KUKA KRL program: MyProgram_228().src

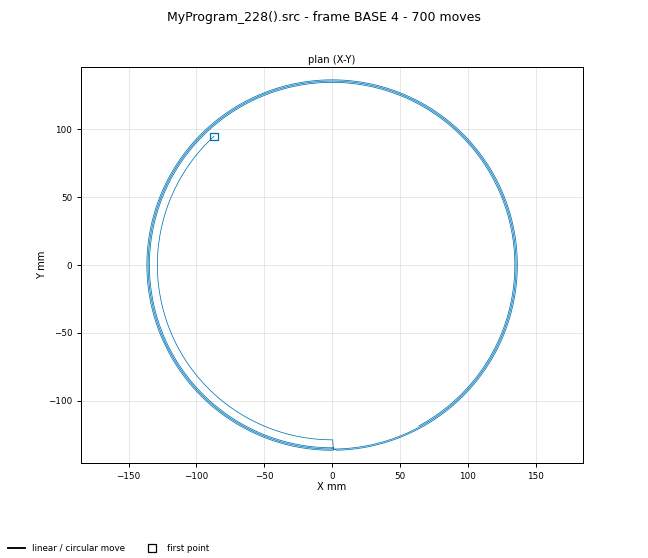
[picture p0: tool path of MyProgram_228().src in frame BASE 4, 700 of 700 moves have a stored position in this frame; points joined in program order, loops and branches not executed]
&ACCESS RVP
&REL 1
&PARAM TEMPLATE = C:\KRC\Roboter\Template\vorgabe
&PARAM EDITMASK = *
DEF MyProgram_228()
; ---- Setting reference (Base) ----
$BASE = BASE_DATA[4]

; --------------------------
; ---- Setting tool (TCP) ----
$TOOL = TOOL_DATA[3]
; --------------------------

$VEL.CP = VEL_APROX_PRINT
Startdeposition()
$VEL.CP = VEL_PRINT
LIN {X -87.249,Y 94.7644,Z 156,A 131.7376,B 16.1467,C -0.3808,E1 16.0419,E2 317.28} C_DIS
LIN {X -90.1231,Y 92.0354,Z 156,A 133.506,B 16.1468,C -0.3771,E1 16.0384,E2 315.5131} C_DIS
LIN {X -93.2907,Y 88.8233,Z 156,A 135.5438,B 16.1468,C -0.3735,E1 16.0344,E2 313.4743} C_DIS
LIN {X -95.9677,Y 85.9237,Z 156,A 137.2975,B 16.147,C -0.3694,E1 16.0311,E2 311.7231} C_DIS
LIN {X -98.5652,Y 82.9313,Z 156,A 139.0194,B 16.1471,C -0.364,E1 16.028,E2 310.008} C_DIS
LIN {X -101.0601,Y 79.8729,Z 156,A 140.9035,B 16.1471,C -0.3635,E1 16.0247,E2 308.1116} C_DIS
LIN {X -103.7403,Y 76.3586,Z 156,A 142.847,B 16.1472,C -0.3579,E1 16.0215,E2 306.1732} C_DIS
LIN {X -106.2189,Y 72.8714,Z 156,A 144.716,B 16.1474,C -0.352,E1 16.0185,E2 304.3107} C_DIS
LIN {X -108.2169,Y 69.8706,Z 156,A 146.2635,B 16.1474,C -0.3462,E1 16.0161,E2 302.7718} C_DIS
LIN {X -109.8979,Y 67.195,Z 156,A 147.6521,B 16.1476,C -0.342,E1 16.0141,E2 301.3869} C_DIS
LIN {X -111.2983,Y 64.8499,Z 156,A 148.8967,B 16.1476,C -0.3396,E1 16.0123,E2 300.1406} C_DIS
LIN {X -112.8404,Y 62.1274,Z 156,A 150.3075,B 16.1476,C -0.3364,E1 16.0104,E2 298.7295} C_DIS
LIN {X -114.5112,Y 58.9894,Z 156,A 151.8787,B 16.1478,C -0.3318,E1 16.0084,E2 297.1616} C_DIS
LIN {X -115.8793,Y 56.2567,Z 156,A 153.2802,B 16.1478,C -0.3292,E1 16.0066,E2 295.7572} C_DIS
LIN {X -117.1898,Y 53.4711,Z 156,A 154.6946,B 16.1478,C -0.3267,E1 16.005,E2 294.3395} C_DIS
LIN {X -118.5677,Y 50.3434,Z 156,A 156.1834,B 16.148,C -0.3214,E1 16.0033,E2 292.8564} C_DIS
LIN {X -119.7652,Y 47.4248,Z 156,A 157.6082,B 16.148,C -0.3181,E1 16.0019,E2 291.4311} C_DIS
LIN {X -120.8905,Y 44.4777,Z 156,A 159.166,B 16.148,C -0.3185,E1 16.0003,E2 289.8575} C_DIS
LIN {X -122.1722,Y 40.8189,Z 156,A 160.8434,B 16.1482,C -0.3121,E1 15.9988,E2 288.1877} C_DIS
LIN {X -123.2669,Y 37.3845,Z 156,A 162.4226,B 16.1482,C -0.3067,E1 15.9975,E2 286.6135} C_DIS
LIN {X -124.267,Y 33.9193,Z 156,A 164.0055,B 16.1484,C -0.3013,E1 15.9963,E2 285.0354} C_DIS
LIN {X -125.2204,Y 30.2007,Z 156,A 165.4905,B 16.1486,C -0.2898,E1 15.9953,E2 283.5781} C_DIS
LIN {X -125.7812,Y 27.7795,Z 156,A 166.7692,B 16.1486,C -0.2915,E1 15.9945,E2 282.2811} C_DIS
LIN {X -126.4236,Y 24.6901,Z 156,A 168.1468,B 16.1486,C -0.2865,E1 15.9938,E2 280.9084} C_DIS
LIN {X -126.9922,Y 21.5728,Z 156,A 169.6871,B 16.1486,C -0.2861,E1 15.993,E2 279.355} C_DIS
LIN {X -127.4822,Y 18.4562,Z 156,A 170.9529,B 16.1488,C -0.2779,E1 15.9925,E2 278.1069} C_DIS
LIN {X -127.8958,Y 15.3281,Z 156,A 172.6093,B 16.1488,C -0.2809,E1 15.9919,E2 276.4233} C_DIS
LIN {X -128.3353,Y 11.0629,Z 156,A 174.5297,B 16.1488,C -0.2755,E1 15.9914,E2 274.504} C_DIS
LIN {X -128.5967,Y 7.4451,Z 156,A 176.2254,B 16.1488,C -0.273,E1 15.9911,E2 272.801} C_DIS
LIN {X -128.7414,Y 4.2996,Z 156,A 177.5163,B 16.149,C -0.2655,E1 15.991,E2 271.5246} C_DIS
LIN {X -128.8029,Y 1.5734,Z 156,A 178.8128,B 16.149,C -0.2643,E1 15.9909,E2 270.22} C_DIS
LIN {X -128.8028,Y -1.5789,Z 156,A -179.8543,B 16.149,C -0.258,E1 15.9909,E2 268.8969} C_DIS
LIN {X -128.7239,Y -4.7473,Z 156,A -178.4414,B 16.1492,C -0.2538,E1 15.991,E2 267.4854} C_DIS
LIN {X -128.5687,Y -7.8985,Z 156,A -176.9705,B 16.1492,C -0.2515,E1 15.9913,E2 266.0085} C_DIS
LIN {X -128.2352,Y -12.1673,Z 156,A -175.3618,B 16.1494,C -0.2372,E1 15.9916,E2 264.4362} C_DIS
LIN {X -127.899,Y -15.3015,Z 156,A -173.6271,B 16.1494,C -0.2426,E1 15.9922,E2 262.665} C_DIS
LIN {X -127.4183,Y -18.9032,Z 156,A -172.0698,B 16.1494,C -0.2361,E1 15.9928,E2 261.1165} C_DIS
LIN {X -126.8381,Y -22.4593,Z 156,A -170.5916,B 16.1495,C -0.2277,E1 15.9935,E2 259.6545} C_DIS
LIN {X -126.2498,Y -25.5591,Z 156,A -169.1609,B 16.1495,C -0.2243,E1 15.9942,E2 258.2223} C_DIS
LIN {X -125.5776,Y -28.6793,Z 156,A -167.594,B 16.1495,C -0.2245,E1 15.9952,E2 256.6402} C_DIS
LIN {X -124.6725,Y -32.3966,Z 156,A -165.7419,B 16.1495,C -0.2239,E1 15.9965,E2 254.7727} C_DIS
LIN {X -123.7153,Y -35.873,Z 156,A -164.1536,B 16.1497,C -0.2188,E1 15.9977,E2 253.1879} C_DIS
LIN {X -122.6587,Y -39.3328,Z 156,A -162.6301,B 16.1497,C -0.2117,E1 15.9989,E2 251.676} C_DIS
LIN {X -121.65,Y -42.3498,Z 156,A -161.112,B 16.1497,C -0.2107,E1 16.0003,E2 250.1475} C_DIS
LIN {X -120.177,Y -46.3659,Z 156,A -159.2834,B 16.1499,C -0.2032,E1 16.0021,E2 248.3295} C_DIS
LIN {X -119.0055,Y -49.2954,Z 156,A -157.8691,B 16.1499,C -0.1997,E1 16.0036,E2 246.9153} C_DIS
LIN {X -117.7369,Y -52.2526,Z 156,A -156.4462,B 16.1499,C -0.1955,E1 16.0052,E2 245.4948} C_DIS
LIN {X -116.4498,Y -55.0627,Z 156,A -155.0417,B 16.1499,C -0.1927,E1 16.0068,E2 244.0882} C_DIS
LIN {X -114.9305,Y -58.1657,Z 156,A -153.4439,B 16.15,C -0.1904,E1 16.0088,E2 242.4848} C_DIS
LIN {X -113.3903,Y -61.1175,Z 156,A -151.9893,B 16.15,C -0.1857,E1 16.0107,E2 241.0347} C_DIS
LIN {X -111.7243,Y -64.113,Z 156,A -150.489,B 16.1501,C -0.1811,E1 16.0128,E2 239.5386} C_DIS
LIN {X -110.1684,Y -66.7504,Z 156,A -148.9834,B 16.1501,C -0.1819,E1 16.015,E2 238.0175} C_DIS
LIN {X -107.9795,Y -70.2361,Z 156,A -147.2344,B 16.1501,C -0.1749,E1 16.0176,E2 236.2795} C_DIS
LIN {X -105.9806,Y -73.2185,Z 156,A -145.4796,B 16.1501,C -0.1758,E1 16.0204,E2 234.5076} C_DIS
LIN {X -103.4626,Y -76.7348,Z 156,A -143.5723,B 16.1502,C -0.1707,E1 16.0235,E2 232.6037} C_DIS
LIN {X -100.9438,Y -80.0194,Z 156,A -141.6939,B 16.1502,C -0.1676,E1 16.0267,E2 230.7223} C_DIS
LIN {X -98.0535,Y -83.5357,Z 156,A -139.6814,B 16.1503,C -0.1627,E1 16.0303,E2 228.7126} C_DIS
LIN {X -95.448,Y -86.5006,Z 156,A -137.9263,B 16.1503,C -0.1589,E1 16.0336,E2 226.9587} C_DIS
LIN {X -93.1464,Y -88.9743,Z 156,A -136.4044,B 16.1503,C -0.1563,E1 16.0365,E2 225.4355} C_DIS
LIN {X -89.9537,Y -92.2016,Z 156,A -134.316,B 16.1503,C -0.1543,E1 16.0407,E2 223.3401} C_DIS
LIN {X -86.9226,Y -95.0644,Z 156,A -132.4884,B 16.1504,C -0.1498,E1 16.0444,E2 221.5167} C_DIS
LIN {X -83.9704,Y -97.6815,Z 156,A -130.7347,B 16.1504,C -0.1465,E1 16.0481,E2 219.7639} C_DIS
LIN {X -80.6634,Y -100.4299,Z 156,A -128.8883,B 16.1505,C -0.141,E1 16.0521,E2 217.9261} C_DIS
LIN {X -77.64,Y -102.7848,Z 156,A -127.2105,B 16.1505,C -0.1373,E1 16.0558,E2 216.2521} C_DIS
LIN {X -74.5444,Y -105.0521,Z 156,A -125.3895,B 16.1505,C -0.138,E1 16.0599,E2 214.4185} C_DIS
LIN {X -71.1886,Y -107.3547,Z 156,A -123.5938,B 16.1505,C -0.1347,E1 16.0641,E2 212.625} C_DIS
LIN {X -68.5545,Y -109.0551,Z 156,A -122.2704,B 16.1505,C -0.1304,E1 16.0672,E2 211.3103} C_DIS
LIN {X -66.2577,Y -110.466,Z 156,A -121.0601,B 16.1505,C -0.129,E1 16.0701,E2 210.099} C_DIS
LIN {X -63.4903,Y -112.0795,Z 156,A -119.6307,B 16.1506,C -0.1272,E1 16.0735,E2 208.6694} C_DIS
LIN {X -60.7258,Y -113.6008,Z 156,A -118.1094,B 16.1506,C -0.129,E1 16.0773,E2 207.1345} C_DIS
LIN {X -57.5236,Y -115.2544,Z 156,A -116.6236,B 16.1506,C -0.1234,E1 16.081,E2 205.6627} C_DIS
LIN {X -54.6526,Y -116.6434,Z 156,A -115.249,B 16.1506,C -0.1203,E1 16.0844,E2 204.2934} C_DIS
LIN {X -51.8174,Y -117.931,Z 156,A -113.8147,B 16.1506,C -0.1203,E1 16.0881,E2 202.8535} C_DIS
LIN {X -48.9638,Y -119.1439,Z 156,A -112.4154,B 16.1506,C -0.1196,E1 16.0917,E2 201.4519} C_DIS
LIN {X -46.1238,Y -120.2711,Z 156,A -111.0448,B 16.1506,C -0.1187,E1 16.0953,E2 200.0799} C_DIS
LIN {X -42.3323,Y -121.6561,Z 156,A -109.172,B 16.1506,C -0.1196,E1 16.1002,E2 198.198} C_DIS
LIN {X -38.3136,Y -122.9825,Z 156,A -107.2264,B 16.1506,C -0.1201,E1 16.1054,E2 196.2449} C_DIS
LIN {X -35.3586,Y -123.8647,Z 156,A -105.9028,B 16.1506,C -0.1176,E1 16.109,E2 194.9268} C_DIS
LIN {X -32.4047,Y -124.6704,Z 156,A -104.4449,B 16.1506,C -0.1198,E1 16.1129,E2 193.4574} C_DIS
LIN {X -29.3446,Y -125.4257,Z 156,A -103.2191,B 16.1507,C -0.1134,E1 16.1162,E2 192.2521} C_DIS
LIN {X -26.6975,Y -126.0148,Z 156,A -101.9339,B 16.1507,C -0.1154,E1 16.1197,E2 190.9574} C_DIS
LIN {X -23.3363,Y -126.6811,Z 156,A -100.4229,B 16.1507,C -0.1143,E1 16.1239,E2 189.4476} C_DIS
LIN {X -20.059,Y -127.2401,Z 156,A -98.9484,B 16.1507,C -0.1137,E1 16.1279,E2 187.9731} C_DIS
LIN {X -15.4689,Y -127.879,Z 156,A -97.1029,B 16.1507,C -0.1062,E1 16.133,E2 186.1525} C_DIS
LIN {X -12.6065,Y -128.1931,Z 156,A -95.5324,B 16.1507,C -0.1154,E1 16.1374,E2 184.5474} C_DIS
LIN {X -9.0242,Y -128.4951,Z 156,A -94.0776,B 16.1507,C -0.1106,E1 16.1414,E2 183.109} C_DIS
LIN {X -5.1896,Y -128.7067,Z 156,A -92.6012,B 16.1507,C -0.1031,E1 16.1455,E2 181.6591} C_DIS
LIN {X -2.7134,Y -128.7839,Z 156,A -91.3422,B 16.1507,C -0.1083,E1 16.1491,E2 180.3813} C_DIS
LIN {X 0.4448,Y -128.8107,Z 156,A -89.7625,B 16.1507,C -0.1142,E1 16.1535,E2 178.7802} C_DIS
LIN {X 0.4448,Y -128.8107,Z 156,A -89.7625,B 16.1507,C -0.1142,E1 16.1535,E2 178.7802} C_DIS
Enddeposition()
LIN {X 0.9577,Y -136.4876,Z 157,A -93.1618,B 24.9717,C -1.2298,E1 24.9996,E2 179.8882} C_DIS
Startdeposition()
$VEL.CP = VEL_PRINT
LIN {X -4.793,Y -136.4624,Z 157,A -95.2992,B 24.9711,C -1.2432,E1 24.9937,E2 181.994} C_DIS
LIN {X -11.5417,Y -136.0568,Z 157,A -97.812,B 24.9702,C -1.2606,E1 24.9869,E2 184.4665} C_DIS
LIN {X -17.4629,Y -135.4244,Z 157,A -100.4347,B 24.9705,C -1.2541,E1 24.9795,E2 187.106} C_DIS
LIN {X -22.0632,Y -134.7517,Z 157,A -102.641,B 24.9712,C -1.241,E1 24.9733,E2 189.3454} C_DIS
LIN {X -25.4466,Y -134.1534,Z 157,A -104.0634,B 24.9711,C -1.2426,E1 24.9694,E2 190.7655} C_DIS
LIN {X -28.8158,Y -133.4701,Z 157,A -105.4664,B 24.971,C -1.2453,E1 24.9656,E2 192.1637} C_DIS
LIN {X -32.1255,Y -132.7124,Z 157,A -106.9209,B 24.971,C -1.2445,E1 24.9617,E2 193.6221} C_DIS
LIN {X -35.9393,Y -131.7329,Z 157,A -108.5566,B 24.971,C -1.2463,E1 24.9572,E2 195.2558} C_DIS
LIN {X -38.9621,Y -130.8698,Z 157,A -109.8853,B 24.9709,C -1.2468,E1 24.9537,E2 196.5856} C_DIS
LIN {X -42.1527,Y -129.8773,Z 157,A -111.2482,B 24.9707,C -1.25,E1 24.9501,E2 197.9434} C_DIS
LIN {X -44.9713,Y -128.9272,Z 157,A -112.5846,B 24.9709,C -1.2464,E1 24.9465,E2 199.2909} C_DIS
LIN {X -48.5684,Y -127.6173,Z 157,A -114.1394,B 24.9707,C -1.2506,E1 24.9425,E2 200.8389} C_DIS
LIN {X -51.6804,Y -126.3889,Z 157,A -115.5554,B 24.9707,C -1.2514,E1 24.9388,E2 202.2561} C_DIS
LIN {X -54.8493,Y -125.0464,Z 157,A -117.0748,B 24.9707,C -1.249,E1 24.9349,E2 203.7847} C_DIS
LIN {X -59.0833,Y -123.1006,Z 157,A -118.9953,B 24.9706,C -1.2532,E1 24.93,E2 205.7001} C_DIS
LIN {X -62.4726,Y -121.4169,Z 157,A -120.5555,B 24.9704,C -1.2567,E1 24.9261,E2 207.2562} C_DIS
LIN {X -65.2945,Y -119.9238,Z 157,A -122.0012,B 24.9706,C -1.253,E1 24.9225,E2 208.7148} C_DIS
LIN {X -69.2384,Y -117.6908,Z 157,A -123.9078,B 24.9705,C -1.2555,E1 24.9179,E2 210.621} C_DIS
LIN {X -73.2088,Y -115.2636,Z 157,A -125.7821,B 24.9701,C -1.2626,E1 24.9135,E2 212.4844} C_DIS
LIN {X -76.368,Y -113.1947,Z 157,A -127.4717,B 24.9703,C -1.2598,E1 24.9096,E2 214.1862} C_DIS
LIN {X -80.1611,Y -110.5408,Z 157,A -129.3474,B 24.97,C -1.2666,E1 24.9053,E2 216.0522} C_DIS
LIN {X -83.5476,Y -108.004,Z 157,A -131.1702,B 24.97,C -1.2674,E1 24.9012,E2 217.8796} C_DIS
LIN {X -87.0681,Y -105.1866,Z 157,A -133.1165,B 24.9699,C -1.2682,E1 24.897,E2 219.8314} C_DIS
LIN {X -90.2129,Y -102.5027,Z 157,A -134.8342,B 24.9697,C -1.2726,E1 24.8934,E2 221.5454} C_DIS
LIN {X -93.618,Y -99.402,Z 157,A -136.7917,B 24.9695,C -1.2753,E1 24.8894,E2 223.5043} C_DIS
LIN {X -96.6303,Y -96.4767,Z 157,A -138.5786,B 24.9695,C -1.2779,E1 24.8858,E2 225.2927} C_DIS
LIN {X -99.9068,Y -93.079,Z 157,A -140.4529,B 24.9689,C -1.2878,E1 24.8823,E2 227.1517} C_DIS
LIN {X -102.6938,Y -89.9952,Z 157,A -142.3091,B 24.969,C -1.2861,E1 24.8788,E2 229.0201} C_DIS
LIN {X -105.7402,Y -86.3949,Z 157,A -144.2944,B 24.9688,C -1.2906,E1 24.8752,E2 231.0039} C_DIS
LIN {X -108.6802,Y -82.6668,Z 157,A -146.2709,B 24.9685,C -1.2963,E1 24.8719,E2 232.9762} C_DIS
LIN {X -111.3396,Y -79.0489,Z 157,A -148.2093,B 24.9685,C -1.2984,E1 24.8687,E2 234.9191} C_DIS
LIN {X -113.7117,Y -75.5962,Z 157,A -149.8638,B 24.9679,C -1.3082,E1 24.8661,E2 236.5584} C_DIS
LIN {X -116.0225,Y -71.9991,Z 157,A -151.7512,B 24.9679,C -1.3082,E1 24.8633,E2 238.4552} C_DIS
LIN {X -118.1139,Y -68.5141,Z 157,A -153.3784,B 24.9675,C -1.3169,E1 24.861,E2 240.0702} C_DIS
LIN {X -120.101,Y -64.9689,Z 157,A -155.2095,B 24.9675,C -1.3153,E1 24.8585,E2 241.9147} C_DIS
LIN {X -124.9697,Y -55.025,Z 157,A -159.7494,B 24.9667,C -1.334,E1 24.8531,E2 246.4348} C_DIS
LIN {X -126.215,Y -52.1021,Z 157,A -161.0965,B 24.9665,C -1.3373,E1 24.8516,E2 247.7815} C_DIS
LIN {X -127.4612,Y -48.9743,Z 157,A -162.5034,B 24.9663,C -1.3418,E1 24.8502,E2 249.1855} C_DIS
LIN {X -128.6336,Y -45.8067,Z 157,A -164.0021,B 24.9663,C -1.3421,E1 24.8487,E2 250.6921} C_DIS
LIN {X -129.9079,Y -42.0571,Z 157,A -165.6808,B 24.966,C -1.3463,E1 24.8473,E2 252.3703} C_DIS
LIN {X -131.1342,Y -38.0593,Z 157,A -167.407,B 24.9657,C -1.3532,E1 24.8459,E2 254.09} C_DIS
LIN {X -132.2625,Y -33.9314,Z 157,A -169.2124,B 24.9654,C -1.3584,E1 24.8446,E2 255.8936} C_DIS
LIN {X -133.166,Y -30.1904,Z 157,A -170.8008,B 24.9651,C -1.3648,E1 24.8436,E2 257.476} C_DIS
LIN {X -133.9535,Y -26.4884,Z 157,A -172.5568,B 24.9653,C -1.3615,E1 24.8426,E2 259.2501} C_DIS
LIN {X -134.6769,Y -22.5112,Z 157,A -174.0908,B 24.9646,C -1.3751,E1 24.8419,E2 260.7609} C_DIS
LIN {X -135.1582,Y -19.4141,Z 157,A -175.4508,B 24.9645,C -1.3771,E1 24.8413,E2 262.1242} C_DIS
LIN {X -135.5862,Y -16.1562,Z 157,A -176.8171,B 24.9642,C -1.3823,E1 24.8408,E2 263.4865} C_DIS
LIN {X -135.9492,Y -12.7499,Z 157,A -178.3678,B 24.9642,C -1.3813,E1 24.8404,E2 265.0486} C_DIS
LIN {X -136.27,Y -8.6741,Z 157,A 179.954,B 24.9639,C -1.3888,E1 24.84,E2 266.719} C_DIS
LIN {X -136.4579,Y -4.9082,Z 157,A 178.3315,B 24.9637,C -1.392,E1 24.8399,E2 268.3437} C_DIS
LIN {X -136.5447,Y -0.6887,Z 157,A 176.589,B 24.9633,C -1.3993,E1 24.8398,E2 270.0794} C_DIS
LIN {X -136.503,Y 3.4288,Z 157,A 174.8401,B 24.9631,C -1.404,E1 24.8398,E2 271.8276} C_DIS
LIN {X -136.3626,Y 7.0678,Z 157,A 173.2663,B 24.9629,C -1.4068,E1 24.8401,E2 273.4042} C_DIS
LIN {X -136.0949,Y 11.0902,Z 157,A 171.5971,B 24.9626,C -1.4135,E1 24.8404,E2 275.0675} C_DIS
LIN {X -135.7642,Y 14.5853,Z 157,A 170.0652,B 24.9625,C -1.4155,E1 24.8408,E2 276.6038} C_DIS
LIN {X -135.2032,Y 19.0993,Z 157,A 168.2113,B 24.962,C -1.4245,E1 24.8415,E2 278.4473} C_DIS
LIN {X -134.686,Y 22.4568,Z 157,A 166.7957,B 24.9617,C -1.4297,E1 24.8421,E2 279.8589} C_DIS
LIN {X -134.0288,Y 26.0984,Z 157,A 165.0936,B 24.9618,C -1.4275,E1 24.843,E2 281.5765} C_DIS
LIN {X -133.0967,Y 30.4938,Z 157,A 163.3198,B 24.9612,C -1.4392,E1 24.8441,E2 283.3329} C_DIS
LIN {X -132.2919,Y 33.8157,Z 157,A 161.8501,B 24.961,C -1.4421,E1 24.8451,E2 284.8042} C_DIS
LIN {X -131.3195,Y 37.4195,Z 157,A 160.1661,B 24.961,C -1.4413,E1 24.8463,E2 286.4998} C_DIS
LIN {X -130.0192,Y 41.7086,Z 157,A 158.4113,B 24.9604,C -1.4536,E1 24.8478,E2 288.2353} C_DIS
LIN {X -128.769,Y 45.4274,Z 157,A 156.7633,B 24.9601,C -1.4588,E1 24.8493,E2 289.8805} C_DIS
LIN {X -127.6672,Y 48.4352,Z 157,A 155.4364,B 24.9599,C -1.4639,E1 24.8506,E2 291.2025} C_DIS
LIN {X -126.5043,Y 51.394,Z 157,A 154.0589,B 24.9597,C -1.466,E1 24.852,E2 292.5829} C_DIS
LIN {X -125.2431,Y 54.3945,Z 157,A 152.684,B 24.9595,C -1.4698,E1 24.8535,E2 293.9563} C_DIS
LIN {X -123.8056,Y 57.5917,Z 157,A 151.1641,B 24.9595,C -1.4719,E1 24.8553,E2 295.4794} C_DIS
LIN {X -122.2195,Y 60.8868,Z 157,A 149.6565,B 24.9591,C -1.4779,E1 24.8571,E2 296.9809} C_DIS
LIN {X -120.7158,Y 63.8151,Z 157,A 148.2867,B 24.9588,C -1.4827,E1 24.8589,E2 298.3466} C_DIS
LIN {X -118.6745,Y 67.5385,Z 157,A 146.4342,B 24.9588,C -1.4845,E1 24.8614,E2 300.2045} C_DIS
LIN {X -116.4781,Y 71.2598,Z 157,A 144.6247,B 24.9584,C -1.49,E1 24.864,E2 302.0102} C_DIS
LIN {X -114.272,Y 74.7472,Z 157,A 142.8205,B 24.9584,C -1.4914,E1 24.8667,E2 303.8202} C_DIS
LIN {X -111.805,Y 78.3892,Z 157,A 140.9498,B 24.9581,C -1.4954,E1 24.8697,E2 305.6906} C_DIS
LIN {X -108.9004,Y 82.3759,Z 157,A 138.7981,B 24.9581,C -1.4971,E1 24.8733,E2 307.8488} C_DIS
LIN {X -106.407,Y 85.5725,Z 157,A 137.1396,B 24.9576,C -1.5038,E1 24.8761,E2 309.4989} C_DIS
LIN {X -103.4241,Y 89.1545,Z 157,A 135.1904,B 24.9573,C -1.5094,E1 24.8796,E2 311.4439} C_DIS
LIN {X -100.3303,Y 92.6228,Z 157,A 133.2038,B 24.9571,C -1.5126,E1 24.8834,E2 313.4316} C_DIS
LIN {X -97.0811,Y 96.023,Z 157,A 131.3563,B 24.9565,C -1.5239,E1 24.8869,E2 315.2602} C_DIS
LIN {X -94.1868,Y 98.8633,Z 157,A 129.5508,B 24.9565,C -1.5228,E1 24.8906,E2 317.0758} C_DIS
LIN {X -90.8799,Y 101.9117,Z 157,A 127.6624,B 24.9563,C -1.5272,E1 24.8945,E2 318.9613} C_DIS
LIN {X -87.5334,Y 104.8001,Z 157,A 125.7574,B 24.9563,C -1.529,E1 24.8985,E2 320.8695} C_DIS
LIN {X -83.9195,Y 107.7158,Z 157,A 123.7927,B 24.956,C -1.5325,E1 24.9028,E2 322.8332} C_DIS
LIN {X -80.6451,Y 110.1884,Z 157,A 122.0698,B 24.9558,C -1.5361,E1 24.9067,E2 324.5536} C_DIS
LIN {X -76.8585,Y 112.8627,Z 157,A 120.1088,B 24.9556,C -1.5393,E1 24.9112,E2 326.5137} C_DIS
LIN {X -73.1617,Y 115.2933,Z 157,A 118.2561,B 24.9554,C -1.5431,E1 24.9155,E2 328.3633} C_DIS
LIN {X -68.7626,Y 117.9701,Z 157,A 116.1991,B 24.9548,C -1.5524,E1 24.9204,E2 330.4045} C_DIS
LIN {X -65.2408,Y 119.9531,Z 157,A 114.3542,B 24.9551,C -1.5479,E1 24.925,E2 332.2654} C_DIS
LIN {X -61.8376,Y 121.7401,Z 157,A 112.8706,B 24.9546,C -1.5572,E1 24.9286,E2 333.7308} C_DIS
LIN {X -58.5691,Y 123.3463,Z 157,A 111.3055,B 24.9546,C -1.5578,E1 24.9325,E2 335.2986} C_DIS
LIN {X -54.9799,Y 124.9899,Z 157,A 109.6879,B 24.9543,C -1.5623,E1 24.9366,E2 336.9095} C_DIS
LIN {X -51.8857,Y 126.3054,Z 157,A 108.2749,B 24.9542,C -1.5642,E1 24.9403,E2 338.3211} C_DIS
LIN {X -48.938,Y 127.4753,Z 157,A 106.9546,B 24.954,C -1.5666,E1 24.9437,E2 339.6385} C_DIS
LIN {X -45.4104,Y 128.7749,Z 157,A 105.3264,B 24.954,C -1.5661,E1 24.948,E2 341.2713} C_DIS
LIN {X -39.7921,Y 130.6185,Z 157,A 102.4437,B 24.9551,C -1.5485,E1 24.9558,E2 344.201} C_DIS
LIN {X -35.8635,Y 131.7532,Z 157,A 101.2031,B 24.9535,C -1.5747,E1 24.959,E2 345.3811} C_DIS
LIN {X -31.739,Y 132.8055,Z 157,A 99.3031,B 24.9538,C -1.5706,E1 24.9641,E2 347.2936} C_DIS
LIN {X -27.807,Y 133.6852,Z 157,A 97.5439,B 24.9539,C -1.5686,E1 24.969,E2 349.0598} C_DIS
LIN {X -23.9531,Y 134.428,Z 157,A 96.0058,B 24.9535,C -1.5755,E1 24.9731,E2 350.5829} C_DIS
LIN {X -20.4003,Y 135.0137,Z 157,A 94.3846,B 24.9538,C -1.5709,E1 24.9776,E2 352.2167} C_DIS
LIN {X -16.3049,Y 135.5685,Z 157,A 92.7506,B 24.9534,C -1.5772,E1 24.9821,E2 353.8369} C_DIS
LIN {X -12.9463,Y 135.9303,Z 157,A 91.3659,B 24.9532,C -1.5796,E1 24.986,E2 355.2166} C_DIS
LIN {X -9.9611,Y 136.1817,Z 157,A 90.0721,B 24.9533,C -1.5783,E1 24.9896,E2 356.5142} C_DIS
LIN {X -5.8338,Y 136.4218,Z 157,A 88.3084,B 24.9533,C -1.5774,E1 24.9945,E2 358.2805} C_DIS
LIN {X -2.1819,Y 136.5282,Z 157,A 86.7838,B 24.9533,C -1.5782,E1 24.9988,E2 359.8032} C_DIS
LIN {X 2.1123,Y 136.5293,Z 157,A 84.9877,B 24.9533,C -1.5789,E1 25.0038,E2 361.5976} C_DIS
LIN {X 5.5829,Y 136.4316,Z 157,A 83.5592,B 24.9532,C -1.5805,E1 25.0077,E2 363.022} C_DIS
LIN {X 9.0201,Y 136.2487,Z 157,A 82.1389,B 24.9532,C -1.5817,E1 25.0117,E2 364.4388} C_DIS
LIN {X 13.0596,Y 135.9195,Z 157,A 80.3851,B 24.9532,C -1.5788,E1 25.0166,E2 366.1985} C_DIS
LIN {X 17.2659,Y 135.4502,Z 157,A 78.5181,B 24.9536,C -1.5736,E1 25.0218,E2 368.0765} C_DIS
LIN {X 21.2759,Y 134.8782,Z 157,A 76.9322,B 24.9533,C -1.5791,E1 25.0261,E2 369.6478} C_DIS
LIN {X 25.3719,Y 134.1677,Z 157,A 75.1742,B 24.9533,C -1.5777,E1 25.031,E2 371.4072} C_DIS
LIN {X 28.6917,Y 133.4969,Z 157,A 73.798,B 24.9533,C -1.5795,E1 25.0347,E2 372.7775} C_DIS
LIN {X 31.9499,Y 132.7547,Z 157,A 72.3085,B 24.9536,C -1.574,E1 25.0388,E2 374.2779} C_DIS
LIN {X 35.7653,Y 131.7794,Z 157,A 70.7388,B 24.9534,C -1.5773,E1 25.043,E2 375.8373} C_DIS
LIN {X 38.7858,Y 130.9215,Z 157,A 69.4317,B 24.9534,C -1.5769,E1 25.0465,E2 377.143} C_DIS
LIN {X 42.2601,Y 129.843,Z 157,A 67.8913,B 24.9535,C -1.5749,E1 25.0506,E2 378.6854} C_DIS
LIN {X 45.2671,Y 128.8246,Z 157,A 66.5598,B 24.9535,C -1.5738,E1 25.0541,E2 380.0169} C_DIS
LIN {X 48.5995,Y 127.6057,Z 157,A 64.5512,B 24.9553,C -1.5444,E1 25.0596,E2 382.0908} C_DIS
LIN {X 52.6492,Y 125.9865,Z 157,A 62.8275,B 24.9551,C -1.5481,E1 25.064,E2 383.8016} C_DIS
LIN {X 56.3669,Y 124.3695,Z 157,A 61.5582,B 24.9539,C -1.5694,E1 25.0671,E2 385.0175} C_DIS
LIN {X 59.3199,Y 122.9876,Z 157,A 60.19,B 24.9539,C -1.5677,E1 25.0705,E2 386.3862} C_DIS
LIN {X 62.3349,Y 121.487,Z 157,A 58.7389,B 24.9542,C -1.5638,E1 25.0741,E2 387.8426} C_DIS
LIN {X 65.6989,Y 119.7032,Z 157,A 57.0549,B 24.9546,C -1.5568,E1 25.0783,E2 389.5383} C_DIS
LIN {X 69.7582,Y 117.3835,Z 157,A 55.1221,B 24.9546,C -1.5555,E1 25.083,E2 391.4683} C_DIS
LIN {X 73.2899,Y 115.2121,Z 157,A 53.3723,B 24.9549,C -1.5521,E1 25.0871,E2 393.2204} C_DIS
LIN {X 76.7311,Y 112.9489,Z 157,A 51.7419,B 24.9547,C -1.5546,E1 25.0909,E2 394.8395} C_DIS
LIN {X 80.1093,Y 110.5784,Z 157,A 49.9765,B 24.955,C -1.5497,E1 25.0949,E2 396.6104} C_DIS
LIN {X 83.6288,Y 107.9412,Z 157,A 48.1433,B 24.9552,C -1.547,E1 25.099,E2 398.4434} C_DIS
LIN {X 87.4314,Y 104.8857,Z 157,A 46.0308,B 24.9556,C -1.5394,E1 25.1036,E2 400.5658} C_DIS
LIN {X 90.6296,Y 102.1343,Z 157,A 44.2759,B 24.9558,C -1.5366,E1 25.1072,E2 402.3202} C_DIS
LIN {X 93.6909,Y 99.3331,Z 157,A 42.5827,B 24.9558,C -1.5356,E1 25.1107,E2 404.0089} C_DIS
LIN {X 96.9729,Y 96.1319,Z 157,A 40.7305,B 24.9558,C -1.5353,E1 25.1144,E2 405.8539} C_DIS
LIN {X 99.7272,Y 93.2718,Z 157,A 38.9751,B 24.9563,C -1.5266,E1 25.1178,E2 407.6222} C_DIS
LIN {X 102.7045,Y 89.9829,Z 157,A 37.1178,B 24.9566,C -1.5225,E1 25.1212,E2 409.481} C_DIS
LIN {X 105.7328,Y 86.404,Z 157,A 35.1671,B 24.9568,C -1.5187,E1 25.1247,E2 411.4318} C_DIS
LIN {X 108.5961,Y 82.7769,Z 157,A 33.267,B 24.9569,C -1.516,E1 25.1279,E2 413.3292} C_DIS
LIN {X 111.2661,Y 79.1519,Z 157,A 31.4015,B 24.9571,C -1.5125,E1 25.131,E2 415.194} C_DIS
LIN {X 114.2499,Y 74.7808,Z 157,A 29.1505,B 24.9576,C -1.5049,E1 25.1345,E2 417.4517} C_DIS
LIN {X 116.7019,Y 70.893,Z 157,A 27.2269,B 24.9579,C -1.5,E1 25.1373,E2 419.3772} C_DIS
LIN {X 119.0827,Y 66.816,Z 157,A 25.2751,B 24.9581,C -1.4961,E1 25.1401,E2 421.328} C_DIS
LIN {X 121.2687,Y 62.7621,Z 157,A 23.4582,B 24.9581,C -1.4971,E1 25.1424,E2 423.133} C_DIS
LIN {X 122.6961,Y 59.9206,Z 157,A 22.1484,B 24.9581,C -1.4947,E1 25.144,E2 424.4415} C_DIS
LIN {X 124.1878,Y 56.7652,Z 157,A 20.6846,B 24.9584,C -1.4904,E1 25.1458,E2 425.9073} C_DIS
LIN {X 125.5712,Y 53.6355,Z 157,A 19.2595,B 24.9586,C -1.4868,E1 25.1474,E2 427.3332} C_DIS
LIN {X 126.864,Y 50.5017,Z 157,A 17.844,B 24.9588,C -1.4829,E1 25.1488,E2 428.75} C_DIS
LIN {X 127.9768,Y 47.6087,Z 157,A 16.5312,B 24.9591,C -1.4783,E1 25.1501,E2 430.0664} C_DIS
LIN {X 129.1023,Y 44.4661,Z 157,A 15.1623,B 24.9591,C -1.4758,E1 25.1514,E2 431.4335} C_DIS
LIN {X 130.3381,Y 40.7083,Z 157,A 13.5123,B 24.9595,C -1.4712,E1 25.1528,E2 433.085} C_DIS
LIN {X 131.4278,Y 37.0321,Z 157,A 11.8734,B 24.9598,C -1.4645,E1 25.1541,E2 434.7304} C_DIS
LIN {X 132.4568,Y 33.166,Z 157,A 10.2401,B 24.96,C -1.4618,E1 25.1552,E2 436.3607} C_DIS
LIN {X 133.2329,Y 29.8976,Z 157,A 8.8572,B 24.9601,C -1.4588,E1 25.1561,E2 437.7426} C_DIS
LIN {X 133.8813,Y 26.8433,Z 157,A 7.5559,B 24.9603,C -1.4551,E1 25.1569,E2 439.045} C_DIS
LIN {X 134.5105,Y 23.492,Z 157,A 6.1367,B 24.9606,C -1.4511,E1 25.1576,E2 440.4652} C_DIS
LIN {X 135.0564,Y 20.1249,Z 157,A 4.7157,B 24.9608,C -1.447,E1 25.1582,E2 441.8875} C_DIS
LIN {X 135.5469,Y 16.4855,Z 157,A 3.1406,B 24.9612,C -1.4401,E1 25.1587,E2 443.4697} C_DIS
LIN {X 135.9178,Y 13.0773,Z 157,A 1.7221,B 24.9613,C -1.4365,E1 25.1591,E2 444.8882} C_DIS
LIN {X 136.2047,Y 9.6454,Z 157,A 0.3251,B 24.9615,C -1.4345,E1 25.1594,E2 446.2818} C_DIS
LIN {X 136.4058,Y 6.2096,Z 157,A -1.1049,B 24.9617,C -1.4305,E1 25.1597,E2 447.7126} C_DIS
LIN {X 136.5246,Y 2.3983,Z 157,A -2.7383,B 24.9621,C -1.4233,E1 25.1597,E2 449.3533} C_DIS
LIN {X 136.5316,Y -1.9768,Z 157,A -4.6461,B 24.9626,C -1.4131,E1 25.1597,E2 451.2737} C_DIS
LIN {X 136.4106,Y -6.1142,Z 157,A -6.3875,B 24.9629,C -1.407,E1 25.1596,E2 453.0191} C_DIS
LIN {X 136.1631,Y -10.2148,Z 157,A -8.0726,B 24.9631,C -1.4035,E1 25.1592,E2 454.7024} C_DIS
LIN {X 135.7449,Y -14.7647,Z 157,A -9.8964,B 24.9631,C -1.4025,E1 25.1587,E2 456.5178} C_DIS
LIN {X 135.2905,Y -18.4845,Z 157,A -11.5827,B 24.9638,C -1.3907,E1 25.1581,E2 458.2219} C_DIS
LIN {X 134.6872,Y -22.4494,Z 157,A -13.1428,B 24.9637,C -1.3922,E1 25.1575,E2 459.7694} C_DIS
LIN {X 134.0986,Y -25.7332,Z 157,A -14.4891,B 24.9637,C -1.3906,E1 25.1568,E2 461.1115} C_DIS
LIN {X 133.465,Y -28.8392,Z 157,A -15.8085,B 24.964,C -1.3869,E1 25.156,E2 462.4321} C_DIS
LIN {X 132.762,Y -31.9197,Z 157,A -17.1315,B 24.9642,C -1.3827,E1 25.1552,E2 463.7573} C_DIS
LIN {X 131.9352,Y -35.181,Z 157,A -18.5636,B 24.9645,C -1.3769,E1 25.1542,E2 465.1948} C_DIS
LIN {X 131.0268,Y -38.426,Z 157,A -19.98,B 24.9647,C -1.3722,E1 25.1531,E2 466.6142} C_DIS
LIN {X 129.8225,Y -42.3243,Z 157,A -21.6638,B 24.9649,C -1.3682,E1 25.1517,E2 468.2978} C_DIS
LIN {X 128.6479,Y -45.767,Z 157,A -23.2355,B 24.9653,C -1.3607,E1 25.1502,E2 469.8783} C_DIS
LIN {X 127.2592,Y -49.494,Z 157,A -24.8018,B 24.9653,C -1.3613,E1 25.1487,E2 471.4345} C_DIS
LIN {X 125.9933,Y -52.633,Z 157,A -26.2722,B 24.9657,C -1.3539,E1 25.1471,E2 472.9141} C_DIS
LIN {X 124.542,Y -55.9811,Z 157,A -27.7736,B 24.9658,C -1.3508,E1 25.1454,E2 474.4146} C_DIS
LIN {X 122.8137,Y -59.6824,Z 157,A -29.4477,B 24.966,C -1.3478,E1 25.1434,E2 476.0869} C_DIS
LIN {X 121.2947,Y -62.7124,Z 157,A -31.0327,B 24.9667,C -1.3342,E1 25.1414,E2 477.6956} C_DIS
LIN {X 119.0126,Y -66.9408,Z 157,A -33.0028,B 24.9668,C -1.3307,E1 25.1387,E2 479.6636} C_DIS
LIN {X 116.9041,Y -70.5585,Z 157,A -34.7192,B 24.967,C -1.3278,E1 25.1363,E2 481.3781} C_DIS
LIN {X 114.8349,Y -73.879,Z 157,A -36.1038,B 24.9665,C -1.3376,E1 25.1342,E2 482.7326} C_DIS
LIN {X 113.0794,Y -76.5384,Z 157,A -37.7118,B 24.9674,C -1.3183,E1 25.1317,E2 484.3779} C_DIS
LIN {X 110.3359,Y -80.4438,Z 157,A -39.7149,B 24.9677,C -1.3126,E1 25.1284,E2 486.3847} C_DIS
LIN {X 107.7895,Y -83.8244,Z 157,A -41.4477,B 24.9679,C -1.3101,E1 25.1255,E2 488.1152} C_DIS
LIN {X 105.1348,Y -87.1306,Z 157,A -43.2122,B 24.968,C -1.3061,E1 25.1224,E2 489.881} C_DIS
LIN {X 102.0741,Y -90.6976,Z 157,A -45.1792,B 24.9683,C -1.3012,E1 25.1188,E2 491.8507} C_DIS
LIN {X 99.1221,Y -93.9146,Z 157,A -47.1407,B 24.9689,C -1.2892,E1 25.115,E2 493.832} C_DIS
LIN {X 95.7314,Y -97.3683,Z 157,A -49.0129,B 24.9687,C -1.293,E1 25.1113,E2 495.6873} C_DIS
LIN {X 92.545,Y -100.4018,Z 157,A -50.8587,B 24.9689,C -1.2885,E1 25.1075,E2 497.5361} C_DIS
LIN {X 89.1452,Y -103.4321,Z 157,A -52.7878,B 24.9692,C -1.283,E1 25.1035,E2 499.4706} C_DIS
LIN {X 86.2008,Y -105.8988,Z 157,A -54.3058,B 24.9691,C -1.2845,E1 25.1002,E2 500.9791} C_DIS
LIN {X 82.862,Y -108.5309,Z 157,A -56.0445,B 24.9691,C -1.2831,E1 25.0964,E2 502.7147} C_DIS
LIN {X 79.539,Y -110.9893,Z 157,A -57.8805,B 24.9696,C -1.2737,E1 25.0922,E2 504.5664} C_DIS
LIN {X 76.0927,Y -113.3803,Z 157,A -59.6433,B 24.9698,C -1.2699,E1 25.0882,E2 506.3323} C_DIS
LIN {X 72.1151,Y -115.9503,Z 157,A -61.5784,B 24.9698,C -1.2689,E1 25.0836,E2 508.2635} C_DIS
LIN {X 68.5232,Y -118.1087,Z 157,A -63.3465,B 24.97,C -1.265,E1 25.0793,E2 510.0354} C_DIS
LIN {X 65.0999,Y -120.0299,Z 157,A -64.9671,B 24.97,C -1.2635,E1 25.0754,E2 511.6548} C_DIS
LIN {X 61.7829,Y -121.7679,Z 157,A -66.4292,B 24.97,C -1.2669,E1 25.0718,E2 513.1048} C_DIS
LIN {X 56.3185,Y -124.3911,Z 157,A -68.9004,B 24.97,C -1.2667,E1 25.0656,E2 515.57} C_DIS
LIN {X 52.2455,Y -126.1552,Z 157,A -70.9607,B 24.9706,C -1.253,E1 25.0602,E2 517.6579} C_DIS
LIN {X 47.8955,Y -127.8694,Z 157,A -72.7817,B 24.9704,C -1.258,E1 25.0555,E2 519.4631} C_DIS
LIN {X 44.8643,Y -128.9642,Z 157,A -74.2065,B 24.9706,C -1.2522,E1 25.0517,E2 520.8987} C_DIS
LIN {X 40.7953,Y -130.311,Z 157,A -75.9362,B 24.9706,C -1.2537,E1 25.0471,E2 522.6216} C_DIS
LIN {X 37.6091,Y -131.266,Z 157,A -77.4609,B 24.971,C -1.245,E1 25.043,E2 524.1643} C_DIS
LIN {X 33.3656,Y -132.4061,Z 157,A -79.187,B 24.9708,C -1.2496,E1 25.0384,E2 525.877} C_DIS
LIN {X 29.3586,Y -133.3529,Z 157,A -80.9387,B 24.9708,C -1.2465,E1 25.0336,E2 527.6334} C_DIS
LIN {X 25.8015,Y -134.0855,Z 157,A -82.4837,B 24.971,C -1.2441,E1 25.0294,E2 529.1824} C_DIS
LIN {X 22.445,Y -134.688,Z 157,A -83.9054,B 24.971,C -1.2434,E1 25.0254,E2 530.6041} C_DIS
LIN {X 18.0176,Y -135.3517,Z 157,A -85.7505,B 24.971,C -1.2439,E1 25.0204,E2 532.4464} C_DIS
LIN {X 14.6126,Y -135.7613,Z 157,A -87.1887,B 24.971,C -1.2431,E1 25.0164,E2 533.8854} C_DIS
LIN {X 10.3003,Y -136.1569,Z 157,A -89.0144,B 24.9711,C -1.2417,E1 25.0113,E2 535.7135} C_DIS
LIN {X 6.6645,Y -136.3829,Z 157,A -90.5059,B 24.9711,C -1.2431,E1 25.0071,E2 537.2013} C_DIS
LIN {X 3.5711,Y -136.499,Z 157,A -93.0366,B 24.9741,C -1.1769,E1 24.9997,E2 539.8881} C_DIS
LIN {X 3.5711,Y -136.499,Z 157,A -93.0366,B 24.9741,C -1.1769,E1 24.9997,E2 539.8881} C_DIS
Enddeposition()
LIN {X 0.9525,Y -135.6041,Z 157,A -92.6752,B 24.9697,C -1.271,E1 25.0013,E2 539.3039} C_DIS
Startdeposition()
$VEL.CP = VEL_PRINT
LIN {X 4.1061,Y -135.5523,Z 157,A -90.8481,B 24.9684,C -1.2981,E1 25.0065,E2 537.4131} C_DIS
LIN {X 8.3057,Y -135.3594,Z 157,A -89.1966,B 24.9687,C -1.292,E1 25.0111,E2 535.7765} C_DIS
LIN {X 11.8908,Y -135.0925,Z 157,A -87.5509,B 24.9684,C -1.2997,E1 25.0157,E2 534.1135} C_DIS
LIN {X 15.8621,Y -134.6832,Z 157,A -85.9687,B 24.9686,C -1.295,E1 25.0201,E2 532.5435} C_DIS
LIN {X 19.5145,Y -134.2029,Z 157,A -84.3273,B 24.9683,C -1.3007,E1 25.0247,E2 530.89} C_DIS
LIN {X 23.846,Y -133.5008,Z 157,A -82.5842,B 24.9685,C -1.2961,E1 25.0294,E2 529.1597} C_DIS
LIN {X 27.2755,Y -132.8428,Z 157,A -81.0315,B 24.9683,C -1.3017,E1 25.0337,E2 527.5957} C_DIS
LIN {X 31.5612,Y -131.8902,Z 157,A -79.2482,B 24.9683,C -1.2995,E1 25.0385,E2 525.8199} C_DIS
LIN {X 37.2296,Y -130.4053,Z 157,A -76.8005,B 24.9683,C -1.3006,E1 25.0451,E2 523.3736} C_DIS
LIN {X 40.72,Y -129.3572,Z 157,A -75.2076,B 24.9681,C -1.3054,E1 25.0494,E2 521.7722} C_DIS
LIN {X 43.9951,Y -128.2797,Z 157,A -73.7429,B 24.968,C -1.3077,E1 25.0533,E2 520.3048} C_DIS
LIN {X 48.6056,Y -126.6051,Z 157,A -71.7185,B 24.968,C -1.3079,E1 25.0586,E2 518.2843} C_DIS
LIN {X 51.9488,Y -125.2696,Z 157,A -70.2098,B 24.9679,C -1.3095,E1 25.0625,E2 516.7753} C_DIS
LIN {X 56.0039,Y -123.5114,Z 157,A -68.359,B 24.9678,C -1.3114,E1 25.0672,E2 514.9245} C_DIS
LIN {X 59.8106,Y -121.7117,Z 157,A -66.8222,B 24.9683,C -1.3009,E1 25.071,E2 513.4164} C_DIS
LIN {X 63.7108,Y -119.7184,Z 157,A -64.6696,B 24.9673,C -1.3209,E1 25.0765,E2 511.2226} C_DIS
LIN {X 67.487,Y -117.6315,Z 157,A -62.915,B 24.9673,C -1.3204,E1 25.0807,E2 509.4744} C_DIS
LIN {X 70.9465,Y -115.5774,Z 157,A -61.1685,B 24.9671,C -1.3263,E1 25.0849,E2 507.7195} C_DIS
LIN {X 74.6604,Y -113.2139,Z 157,A -59.3115,B 24.9669,C -1.3298,E1 25.0893,E2 505.8601} C_DIS
LIN {X 78.2833,Y -110.7398,Z 157,A -57.4662,B 24.9667,C -1.3332,E1 25.0935,E2 504.0131} C_DIS
LIN {X 81.8656,Y -108.1185,Z 157,A -55.56,B 24.9664,C -1.339,E1 25.0978,E2 502.1001} C_DIS
LIN {X 85.3274,Y -105.4079,Z 157,A -53.7972,B 24.9664,C -1.3378,E1 25.1016,E2 500.3467} C_DIS
LIN {X 88.7658,Y -102.5289,Z 157,A -51.7164,B 24.9657,C -1.3528,E1 25.1061,E2 498.2387} C_DIS
LIN {X 92.5748,Y -99.1035,Z 157,A -49.7117,B 24.9659,C -1.349,E1 25.1102,E2 496.2512} C_DIS
LIN {X 95.8035,Y -95.9861,Z 157,A -48.0436,B 24.9663,C -1.3408,E1 25.1135,E2 494.6094} C_DIS
LIN {X 97.902,Y -93.844,Z 157,A -46.4302,B 24.9652,C -1.3636,E1 25.1167,E2 492.9489} C_DIS
LIN {X 101.0673,Y -90.4265,Z 157,A -44.5913,B 24.9652,C -1.3614,E1 25.1201,E2 491.1234} C_DIS
LIN {X 104.0756,Y -86.9477,Z 157,A -42.638,B 24.965,C -1.3672,E1 25.1236,E2 489.1654} C_DIS
LIN {X 106.8486,Y -83.5166,Z 157,A -40.8143,B 24.9648,C -1.37,E1 25.1268,E2 487.3436} C_DIS
LIN {X 109.9688,Y -79.3629,Z 157,A -38.6158,B 24.9645,C -1.3764,E1 25.1305,E2 485.1406} C_DIS
LIN {X 112.3936,Y -75.8898,Z 157,A -36.8898,B 24.9645,C -1.3779,E1 25.1332,E2 483.4195} C_DIS
LIN {X 114.6369,Y -72.4564,Z 157,A -35.1019,B 24.964,C -1.3861,E1 25.1359,E2 481.6213} C_DIS
LIN {X 117.0841,Y -68.4322,Z 157,A -33.1264,B 24.9637,C -1.3912,E1 25.1387,E2 479.644} C_DIS
LIN {X 119.2342,Y -64.6135,Z 157,A -31.2765,B 24.9635,C -1.3967,E1 25.1412,E2 477.7908} C_DIS
LIN {X 120.9321,Y -61.3715,Z 157,A -29.8494,B 24.9635,C -1.3946,E1 25.143,E2 476.3761} C_DIS
LIN {X 122.5446,Y -58.0862,Z 157,A -28.2375,B 24.9631,C -1.4032,E1 25.145,E2 474.7527} C_DIS
LIN {X 123.9302,Y -55.0675,Z 157,A -26.321,B 24.9613,C -1.437,E1 25.1473,E2 472.7668} C_DIS
LIN {X 125.8388,Y -50.5535,Z 157,A -25.1571,B 24.9637,C -1.3915,E1 25.1484,E2 471.7165} C_DIS
LIN {X 127.1978,Y -47.0329,Z 157,A -23.1468,B 24.9622,C -1.4203,E1 25.1504,E2 469.6496} C_DIS
LIN {X 128.5702,Y -43.1375,Z 157,A -21.3699,B 24.9618,C -1.4278,E1 25.152,E2 467.8651} C_DIS
LIN {X 130.0668,Y -38.3898,Z 157,A -19.4574,B 24.962,C -1.4237,E1 25.1536,E2 465.9732} C_DIS
LIN {X 130.9924,Y -35.1011,Z 157,A -18.0146,B 24.9618,C -1.4284,E1 25.1546,E2 464.5276} C_DIS
LIN {X 131.8072,Y -31.9054,Z 157,A -16.6323,B 24.9616,C -1.4323,E1 25.1556,E2 463.1441} C_DIS
LIN {X 132.5678,Y -28.5811,Z 157,A -15.218,B 24.9614,C -1.4355,E1 25.1564,E2 461.7305} C_DIS
LIN {X 133.2192,Y -25.3721,Z 157,A -13.7934,B 24.961,C -1.4424,E1 25.1572,E2 460.2978} C_DIS
LIN {X 133.9703,Y -21.0513,Z 157,A -11.932,B 24.9607,C -1.449,E1 25.158,E2 458.4318} C_DIS
LIN {X 134.5132,Y -17.2475,Z 157,A -10.2683,B 24.9602,C -1.4567,E1 25.1587,E2 456.7598} C_DIS
LIN {X 134.9873,Y -13.0216,Z 157,A -8.5693,B 24.9602,C -1.4571,E1 25.1592,E2 455.0699} C_DIS
LIN {X 135.3249,Y -8.8666,Z 157,A -6.7882,B 24.9598,C -1.4641,E1 25.1595,E2 453.2829} C_DIS
LIN {X 135.5152,Y -5.1783,Z 157,A -5.2647,B 24.9597,C -1.4672,E1 25.1597,E2 451.7612} C_DIS
LIN {X 135.6124,Y -0.8057,Z 157,A -3.4759,B 24.9595,C -1.4699,E1 25.1597,E2 449.9766} C_DIS
LIN {X 135.5818,Y 3.0452,Z 157,A -1.7214,B 24.9588,C -1.4826,E1 25.1597,E2 448.2026} C_DIS
LIN {X 135.4213,Y 7.2404,Z 157,A 0.0174,B 24.9586,C -1.4865,E1 25.1595,E2 446.4651} C_DIS
LIN {X 135.1291,Y 11.4572,Z 157,A 1.7111,B 24.9586,C -1.4871,E1 25.1591,E2 444.7799} C_DIS
LIN {X 134.7021,Y 15.7034,Z 157,A 3.503,B 24.9583,C -1.4924,E1 25.1586,E2 442.9862} C_DIS
LIN {X 134.2544,Y 19.1538,Z 157,A 4.9319,B 24.9581,C -1.4948,E1 25.158,E2 441.5599} C_DIS
LIN {X 133.7364,Y 22.4879,Z 157,A 6.3681,B 24.9578,C -1.5001,E1 25.1574,E2 440.1198} C_DIS
LIN {X 132.9705,Y 26.648,Z 157,A 8.1964,B 24.9574,C -1.5082,E1 25.1564,E2 438.2832} C_DIS
LIN {X 132.1946,Y 30.2603,Z 157,A 9.658,B 24.9574,C -1.5075,E1 25.1556,E2 436.8316} C_DIS
LIN {X 131.4152,Y 33.4836,Z 157,A 11.0679,B 24.9571,C -1.5124,E1 25.1546,E2 435.4183} C_DIS
LIN {X 130.4838,Y 36.9491,Z 157,A 12.426,B 24.9574,C -1.5082,E1 25.1536,E2 434.0779} C_DIS
LIN {X 129.3534,Y 40.7316,Z 157,A 14.315,B 24.9564,C -1.526,E1 25.1521,E2 432.1578} C_DIS
LIN {X 128.1616,Y 44.3357,Z 157,A 15.9348,B 24.956,C -1.5318,E1 25.1506,E2 430.5334} C_DIS
LIN {X 126.5412,Y 48.7701,Z 157,A 17.7943,B 24.9561,C -1.5302,E1 25.1488,E2 428.6881} C_DIS
LIN {X 125.2387,Y 52.0227,Z 157,A 19.2818,B 24.9559,C -1.535,E1 25.1472,E2 427.1974} C_DIS
LIN {X 123.8294,Y 55.293,Z 157,A 20.7699,B 24.9557,C -1.5386,E1 25.1455,E2 425.7091} C_DIS
LIN {X 120.9373,Y 61.3613,Z 157,A 23.6204,B 24.9551,C -1.5473,E1 25.1421,E2 422.8532} C_DIS
LIN {X 119.3037,Y 64.4848,Z 157,A 25.167,B 24.9547,C -1.5547,E1 25.14,E2 421.2972} C_DIS
LIN {X 117.1011,Y 68.4032,Z 157,A 27.0977,B 24.9543,C -1.5618,E1 25.1373,E2 419.3599} C_DIS
LIN {X 114.7122,Y 72.3372,Z 157,A 29.0044,B 24.9541,C -1.5649,E1 25.1345,E2 417.4555} C_DIS
LIN {X 110.8477,Y 78.1303,Z 157,A 32.1439,B 24.953,C -1.5838,E1 25.1295,E2 414.2871} C_DIS
LIN {X 108.8583,Y 80.8792,Z 157,A 33.3585,B 24.9535,C -1.5751,E1 25.1276,E2 413.0987} C_DIS
LIN {X 106.0047,Y 84.5847,Z 157,A 35.3172,B 24.9533,C -1.579,E1 25.1242,E2 411.14} C_DIS
LIN {X 103.102,Y 88.1001,Z 157,A 37.2467,B 24.953,C -1.5838,E1 25.1207,E2 409.208} C_DIS
LIN {X 100.1255,Y 91.4692,Z 157,A 39.1456,B 24.9527,C -1.5882,E1 25.1172,E2 407.3071} C_DIS
LIN {X 97.2279,Y 94.5429,Z 157,A 40.923,B 24.9525,C -1.5919,E1 25.1137,E2 405.5289} C_DIS
LIN {X 94.0189,Y 97.7353,Z 157,A 42.8369,B 24.9523,C -1.5961,E1 25.1099,E2 403.613} C_DIS
LIN {X 90.9022,Y 100.6401,Z 157,A 44.6023,B 24.9522,C -1.5979,E1 25.1063,E2 401.8504} C_DIS
LIN {X 87.5259,Y 103.5902,Z 157,A 46.2282,B 24.9528,C -1.5869,E1 25.1029,E2 400.2569} C_DIS
LIN {X 84.013,Y 106.4584,Z 157,A 48.4988,B 24.9514,C -1.6102,E1 25.0979,E2 397.9399} C_DIS
LIN {X 80.0848,Y 109.4442,Z 157,A 50.4681,B 24.9516,C -1.6076,E1 25.0935,E2 395.9838} C_DIS
LIN {X 76.3692,Y 112.069,Z 157,A 52.4256,B 24.9513,C -1.6128,E1 25.089,E2 394.0205} C_DIS
LIN {X 72.5233,Y 114.5947,Z 157,A 54.3289,B 24.9513,C -1.6138,E1 25.0845,E2 392.1212} C_DIS
LIN {X 70.1052,Y 116.0897,Z 157,A 55.7807,B 24.9503,C -1.6294,E1 25.081,E2 390.637} C_DIS
LIN {X 66.961,Y 117.9315,Z 157,A 57.0049,B 24.9512,C -1.6143,E1 25.0781,E2 389.4521} C_DIS
LIN {X 63.6342,Y 119.7586,Z 157,A 58.6356,B 24.9509,C -1.6181,E1 25.0741,E2 387.8172} C_DIS
LIN {X 60.2704,Y 121.4849,Z 157,A 60.1594,B 24.9511,C -1.6162,E1 25.0703,E2 386.3021} C_DIS
LIN {X 57.3024,Y 122.9131,Z 157,A 61.5501,B 24.951,C -1.6178,E1 25.0668,E2 384.911} C_DIS
LIN {X 54.6047,Y 124.1362,Z 157,A 62.7723,B 24.951,C -1.6177,E1 25.0637,E2 383.6921} C_DIS
LIN {X 51.5301,Y 125.4444,Z 157,A 64.2815,B 24.9505,C -1.6245,E1 25.0598,E2 382.1703} C_DIS
LIN {X 47.7524,Y 126.9283,Z 157,A 65.9039,B 24.9507,C -1.6213,E1 25.0556,E2 380.5592} C_DIS
LIN {X 43.6257,Y 128.4076,Z 157,A 67.9055,B 24.9502,C -1.631,E1 25.0502,E2 378.5386} C_DIS
LIN {X 40.2256,Y 129.5117,Z 157,A 69.3412,B 24.9503,C -1.6282,E1 25.0464,E2 377.1121} C_DIS
LIN {X 36.5181,Y 130.6043,Z 157,A 70.8515,B 24.9507,C -1.6228,E1 25.0424,E2 375.6171} C_DIS
LIN {X 33.3069,Y 131.46,Z 157,A 72.2885,B 24.9505,C -1.6254,E1 25.0385,E2 374.1761} C_DIS
LIN {X 29.8706,Y 132.2836,Z 157,A 73.8746,B 24.9501,C -1.6313,E1 25.0342,E2 372.5784} C_DIS
LIN {X 25.7161,Y 133.1535,Z 157,A 75.5848,B 24.9504,C -1.6276,E1 25.0295,E2 370.8789} C_DIS
LIN {X 22.3316,Y 133.7625,Z 157,A 77.0343,B 24.9504,C -1.628,E1 25.0255,E2 369.43} C_DIS
LIN {X 18.8425,Y 134.2989,Z 157,A 78.6039,B 24.9501,C -1.6326,E1 25.0212,E2 367.8509} C_DIS
LIN {X 14.6889,Y 134.8162,Z 157,A 80.3016,B 24.9503,C -1.6292,E1 25.0165,E2 366.1626} C_DIS
LIN {X 10.9087,Y 135.1755,Z 157,A 81.9999,B 24.95,C -1.6343,E1 25.0117,E2 364.4531} C_DIS
LIN {X 6.7598,Y 135.4454,Z 157,A 83.6877,B 24.9502,C -1.6307,E1 25.0071,E2 362.7746} C_DIS
LIN {X 2.5286,Y 135.5908,Z 157,A 85.4687,B 24.9502,C -1.63,E1 25.0021,E2 360.9954} C_DIS
LIN {X -1.3425,Y 135.6087,Z 157,A 87.1945,B 24.9499,C -1.6345,E1 24.9972,E2 359.2592} C_DIS
LIN {X -5.2863,Y 135.511,Z 157,A 88.7686,B 24.9503,C -1.6291,E1 24.9929,E2 357.6975} C_DIS
LIN {X -9.459,Y 135.2843,Z 157,A 90.5432,B 24.9503,C -1.6289,E1 24.9879,E2 355.923} C_DIS
LIN {X -13.0271,Y 134.9868,Z 157,A 92.024,B 24.9504,C -1.6264,E1 24.9838,E2 354.4472} C_DIS
LIN {X -16.9494,Y 134.5522,Z 157,A 93.7993,B 24.9501,C -1.6311,E1 24.9789,E2 352.6595} C_DIS
LIN {X -20.7553,Y 134.0162,Z 157,A 95.319,B 24.9505,C -1.6246,E1 24.9747,E2 351.1541} C_DIS
LIN {X -24.4195,Y 133.3982,Z 157,A 97.0019,B 24.9503,C -1.6293,E1 24.9701,E2 349.4584} C_DIS
LIN {X -28.4528,Y 132.5955,Z 157,A 98.6288,B 24.9507,C -1.622,E1 24.9656,E2 347.8468} C_DIS
LIN {X -31.9608,Y 131.7939,Z 157,A 100.1997,B 24.9507,C -1.6232,E1 24.9614,E2 346.271} C_DIS
LIN {X -35.6567,Y 130.8442,Z 157,A 101.7403,B 24.951,C -1.6178,E1 24.9572,E2 344.741} C_DIS
LIN {X -38.295,Y 130.0946,Z 157,A 102.9189,B 24.951,C -1.6175,E1 24.9541,E2 343.5609} C_DIS
LIN {X -42.151,Y 128.8987,Z 157,A 104.6993,B 24.9509,C -1.6194,E1 24.9493,E2 341.7731} C_DIS
LIN {X -45.7508,Y 127.6635,Z 157,A 106.2466,B 24.9512,C -1.6142,E1 24.9453,E2 340.235} C_DIS
LIN {X -48.9306,Y 126.4788,Z 157,A 107.6655,B 24.9513,C -1.6115,E1 24.9416,E2 338.8195} C_DIS
LIN {X -52.0518,Y 125.2266,Z 157,A 109.1218,B 24.9513,C -1.6113,E1 24.9378,E2 337.3605} C_DIS
LIN {X -55.2071,Y 123.8678,Z 157,A 110.5664,B 24.9515,C -1.6087,E1 24.9341,E2 335.9186} C_DIS
LIN {X -58.2521,Y 122.4653,Z 157,A 112.0165,B 24.9515,C -1.6082,E1 24.9304,E2 334.466} C_DIS
LIN {X -61.2362,Y 121.001,Z 157,A 113.3738,B 24.9518,C -1.6035,E1 24.9271,E2 333.1164} C_DIS
LIN {X -64.3169,Y 119.3939,Z 157,A 114.9599,B 24.9516,C -1.607,E1 24.9231,E2 331.5175} C_DIS
LIN {X -68.3157,Y 117.1525,Z 157,A 116.9197,B 24.9518,C -1.6046,E1 24.9184,E2 329.5575} C_DIS
LIN {X -73.2466,Y 114.1337,Z 157,A 119.091,B 24.9529,C -1.5861,E1 24.9133,E2 327.4235} C_DIS
LIN {X -76.6188,Y 111.8978,Z 157,A 121.0253,B 24.9524,C -1.5941,E1 24.9088,E2 325.4638} C_DIS
LIN {X -80.0242,Y 109.4879,Z 157,A 122.8399,B 24.9524,C -1.593,E1 24.9046,E2 323.6453} C_DIS
LIN {X -83.7553,Y 106.6612,Z 157,A 124.7936,B 24.9528,C -1.5875,E1 24.9003,E2 321.6976} C_DIS
LIN {X -86.9419,Y 104.0804,Z 157,A 126.5777,B 24.9528,C -1.5862,E1 24.8965,E2 319.9098} C_DIS
LIN {X -89.1122,Y 102.2281,Z 157,A 127.9606,B 24.9525,C -1.5924,E1 24.8935,E2 318.5068} C_DIS
LIN {X -93.4463,Y 98.2825,Z 157,A 130.2777,B 24.9533,C -1.5784,E1 24.8888,E2 316.2136} C_DIS
LIN {X -96.3792,Y 95.4078,Z 157,A 132.034,B 24.9535,C -1.5752,E1 24.8853,E2 314.4576} C_DIS
LIN {X -100.4047,Y 91.1617,Z 157,A 134.8973,B 24.9527,C -1.5887,E1 24.8798,E2 311.5496} C_DIS
LIN {X -103.2118,Y 87.9711,Z 157,A 136.3024,B 24.9542,C -1.5642,E1 24.8774,E2 310.1964} C_DIS
LIN {X -105.9187,Y 84.6928,Z 157,A 138.1522,B 24.9542,C -1.562,E1 24.8741,E2 308.3431} C_DIS
LIN {X -108.4155,Y 81.4721,Z 157,A 139.7031,B 24.9551,C -1.5487,E1 24.8715,E2 306.8165} C_DIS
LIN {X -110.7128,Y 78.3215,Z 157,A 141.5172,B 24.9548,C -1.5524,E1 24.8685,E2 304.9847} C_DIS
LIN {X -113.2405,Y 74.62,Z 157,A 143.4199,B 24.9551,C -1.5475,E1 24.8656,E2 303.0843} C_DIS
LIN {X -115.7173,Y 70.7185,Z 157,A 145.3556,B 24.9555,C -1.5409,E1 24.8627,E2 301.1544} C_DIS
LIN {X -117.9906,Y 66.8575,Z 157,A 147.3171,B 24.9556,C -1.5387,E1 24.86,E2 299.1878} C_DIS
LIN {X -120.0324,Y 63.1129,Z 157,A 149.0021,B 24.9563,C -1.5275,E1 24.8578,E2 297.5207} C_DIS
LIN {X -121.599,Y 60.0391,Z 157,A 150.4712,B 24.9565,C -1.5236,E1 24.856,E2 296.0529} C_DIS
LIN {X -123.0998,Y 56.8988,Z 157,A 151.9405,B 24.9568,C -1.519,E1 24.8542,E2 294.5865} C_DIS
LIN {X -124.412,Y 53.9695,Z 157,A 153.2982,B 24.957,C -1.5149,E1 24.8527,E2 293.2313} C_DIS
LIN {X -125.6624,Y 50.9911,Z 157,A 154.7123,B 24.9571,C -1.5131,E1 24.8512,E2 291.8137} C_DIS
LIN {X -126.9223,Y 47.7683,Z 157,A 156.1394,B 24.9575,C -1.5067,E1 24.8498,E2 290.3936} C_DIS
LIN {X -128.2309,Y 44.136,Z 157,A 158.4279,B 24.9559,C -1.5344,E1 24.8476,E2 288.0261} C_DIS
LIN {X -129.7682,Y 39.3875,Z 157,A 159.9602,B 24.9579,C -1.4987,E1 24.8464,E2 286.5701} C_DIS
LIN {X -130.9223,Y 35.364,Z 157,A 161.7492,B 24.9582,C -1.494,E1 24.8451,E2 284.782} C_DIS
LIN {X -131.8134,Y 31.8797,Z 157,A 163.5761,B 24.9576,C -1.5044,E1 24.8438,E2 282.9196} C_DIS
LIN {X -132.5877,Y 28.4887,Z 157,A 164.7744,B 24.9586,C -1.486,E1 24.8431,E2 281.7581} C_DIS
LIN {X -133.4447,Y 24.1597,Z 157,A 166.5967,B 24.9591,C -1.4778,E1 24.8422,E2 279.9446} C_DIS
LIN {X -134.0022,Y 20.8458,Z 157,A 168.0482,B 24.9593,C -1.4746,E1 24.8415,E2 278.4919} C_DIS
LIN {X -134.5234,Y 17.1696,Z 157,A 169.6995,B 24.9593,C -1.4736,E1 24.8409,E2 276.8333} C_DIS
LIN {X -134.9708,Y 13.1941,Z 157,A 171.3255,B 24.9598,C -1.4648,E1 24.8404,E2 275.2186} C_DIS
LIN {X -135.2689,Y 9.6699,Z 157,A 172.8744,B 24.9599,C -1.4625,E1 24.8401,E2 273.6656} C_DIS
LIN {X -135.506,Y 5.4133,Z 157,A 174.6461,B 24.9603,C -1.4551,E1 24.8399,E2 271.9011} C_DIS
LIN {X -135.6086,Y 1.3794,Z 157,A 176.4068,B 24.9605,C -1.4522,E1 24.8398,E2 270.1366} C_DIS
LIN {X -135.5848,Y -2.8884,Z 157,A 178.2908,B 24.9605,C -1.4503,E1 24.8398,E2 268.2459} C_DIS
LIN {X -135.4306,Y -7.0552,Z 157,A -179.9792,B 24.961,C -1.4429,E1 24.8401,E2 266.523} C_DIS
LIN {X -135.1418,Y -11.3072,Z 157,A -178.2146,B 24.9614,C -1.4352,E1 24.8405,E2 264.7662} C_DIS
LIN {X -134.7386,Y -15.398,Z 157,A -176.3877,B 24.9614,C -1.434,E1 24.841,E2 262.9312} C_DIS
LIN {X -134.2502,Y -19.1834,Z 157,A -174.8858,B 24.9621,C -1.4232,E1 24.8416,E2 261.4459} C_DIS
LIN {X -133.71,Y -22.6461,Z 157,A -173.5353,B 24.9627,C -1.4119,E1 24.8421,E2 260.1143} C_DIS
LIN {X -132.2126,Y -30.1813,Z 157,A -170.099,B 24.9627,C -1.411,E1 24.8441,E2 256.66} C_DIS
LIN {X -131.3297,Y -33.8201,Z 157,A -168.3954,B 24.9627,C -1.4121,E1 24.8452,E2 254.944} C_DIS
LIN {X -129.8921,Y -38.9826,Z 157,A -166.1257,B 24.963,C -1.4052,E1 24.847,E2 252.6773} C_DIS
LIN {X -128.7525,Y -42.5902,Z 157,A -164.6218,B 24.9635,C -1.3956,E1 24.8483,E2 251.1877} C_DIS
LIN {X -127.6573,Y -45.768,Z 157,A -163.2087,B 24.9638,C -1.3909,E1 24.8496,E2 249.7778} C_DIS
LIN {X -126.4707,Y -48.9515,Z 157,A -161.7588,B 24.9639,C -1.3873,E1 24.851,E2 248.3284} C_DIS
LIN {X -125.2241,Y -52.0578,Z 157,A -160.3352,B 24.9641,C -1.3836,E1 24.8525,E2 246.9057} C_DIS
LIN {X -123.0932,Y -56.913,Z 157,A -157.6791,B 24.9634,C -1.3981,E1 24.8556,E2 244.2006} C_DIS
LIN {X -121.3925,Y -60.4577,Z 157,A -156.3255,B 24.9644,C -1.3777,E1 24.8573,E2 242.8882} C_DIS
LIN {X -119.3462,Y -64.4057,Z 157,A -154.4372,B 24.9647,C -1.3728,E1 24.8597,E2 241.0014} C_DIS
LIN {X -117.1973,Y -68.2383,Z 157,A -152.5466,B 24.9649,C -1.3694,E1 24.8624,E2 239.109} C_DIS
LIN {X -114.8919,Y -72.0524,Z 157,A -150.6504,B 24.9651,C -1.365,E1 24.8651,E2 237.2137} C_DIS
LIN {X -112.5357,Y -75.6798,Z 157,A -148.8005,B 24.9653,C -1.3613,E1 24.868,E2 235.3633} C_DIS
LIN {X -109.951,Y -79.3876,Z 157,A -146.9111,B 24.9656,C -1.3554,E1 24.871,E2 233.4788} C_DIS
LIN {X -106.839,Y -83.5289,Z 157,A -144.7165,B 24.9659,C -1.3502,E1 24.8748,E2 231.286} C_DIS
LIN {X -104.2128,Y -86.7836,Z 157,A -142.9918,B 24.9662,C -1.3438,E1 24.8778,E2 229.5686} C_DIS
LIN {X -101.2247,Y -90.2507,Z 157,A -140.9621,B 24.9662,C -1.3442,E1 24.8816,E2 227.5288} C_DIS
LIN {X -98.1224,Y -93.6138,Z 157,A -139.052,B 24.9664,C -1.3386,E1 24.8852,E2 225.6236} C_DIS
LIN {X -95.0606,Y -96.7215,Z 157,A -137.2055,B 24.9666,C -1.3348,E1 24.8888,E2 223.7785} C_DIS
LIN {X -91.8753,Y -99.7522,Z 157,A -135.3182,B 24.9667,C -1.3324,E1 24.8927,E2 221.8891} C_DIS
LIN {X -88.4308,Y -102.818,Z 157,A -133.3938,B 24.967,C -1.3272,E1 24.8967,E2 219.9694} C_DIS
LIN {X -85.0501,Y -105.6316,Z 157,A -131.5206,B 24.9671,C -1.3244,E1 24.9008,E2 218.0958} C_DIS
LIN {X -81.4139,Y -108.4594,Z 157,A -129.5397,B 24.9672,C -1.3227,E1 24.9052,E2 216.1119} C_DIS
LIN {X -77.826,Y -111.0623,Z 157,A -127.6523,B 24.9674,C -1.3202,E1 24.9095,E2 214.2238} C_DIS
LIN {X -74.2081,Y -113.5116,Z 157,A -125.9414,B 24.9679,C -1.3101,E1 24.9134,E2 212.5312} C_DIS
LIN {X -69.0105,Y -116.7444,Z 157,A -123.2061,B 24.9677,C -1.3139,E1 24.92,E2 209.7785} C_DIS
LIN {X -64.6388,Y -119.2204,Z 157,A -121.0689,B 24.9677,C -1.3117,E1 24.9252,E2 207.6403} C_DIS
LIN {X -60.7757,Y -121.2354,Z 157,A -119.2168,B 24.9679,C -1.3099,E1 24.9298,E2 205.7875} C_DIS
LIN {X -57.4495,Y -122.8451,Z 157,A -117.6542,B 24.9679,C -1.3081,E1 24.9337,E2 204.2253} C_DIS
LIN {X -53.9546,Y -124.4184,Z 157,A -116.1607,B 24.9684,C -1.2996,E1 24.9375,E2 202.7482} C_DIS
LIN {X -50.8637,Y -125.7138,Z 157,A -114.6988,B 24.9684,C -1.3006,E1 24.9413,E2 201.2808} C_DIS
LIN {X -46.336,Y -127.4525,Z 157,A -112.6469,B 24.9684,C -1.2988,E1 24.9467,E2 199.2289} C_DIS
LIN {X -43.4185,Y -128.4766,Z 157,A -111.2876,B 24.9684,C -1.3004,E1 24.9503,E2 197.8631} C_DIS
LIN {X -39.8482,Y -129.6272,Z 157,A -109.797,B 24.9686,C -1.2942,E1 24.9542,E2 196.3846} C_DIS
LIN {X -36.6304,Y -130.573,Z 157,A -108.3532,B 24.9686,C -1.2947,E1 24.9581,E2 194.9374} C_DIS
LIN {X -33.3268,Y -131.455,Z 157,A -106.9108,B 24.9686,C -1.2937,E1 24.962,E2 193.4952} C_DIS
LIN {X -29.4478,Y -132.3802,Z 157,A -105.1033,B 24.9684,C -1.2993,E1 24.967,E2 191.672} C_DIS
LIN {X -25.4973,Y -133.1953,Z 157,A -103.5282,B 24.9687,C -1.2917,E1 24.9712,E2 190.1131} C_DIS
LIN {X -21.9211,Y -133.831,Z 157,A -101.882,B 24.9685,C -1.2972,E1 24.9758,E2 188.4523} C_DIS
LIN {X -17.7527,Y -134.447,Z 157,A -100.2373,B 24.9689,C -1.2895,E1 24.9803,E2 186.8246} C_DIS
LIN {X -14.6228,Y -134.8233,Z 157,A -98.8416,B 24.9687,C -1.2928,E1 24.9842,E2 185.4203} C_DIS
LIN {X -10.9564,Y -135.1714,Z 157,A -97.0613,B 24.9681,C -1.3048,E1 24.9892,E2 183.6107} C_DIS
LIN {X -5.5121,Y -135.5021,Z 157,A -95.0637,B 24.9689,C -1.2883,E1 24.9947,E2 181.6515} C_DIS
LIN {X -0.5772,Y -135.613,Z 157,A -92.7468,B 24.9683,C -1.3013,E1 25.0013,E2 179.3039} C_DIS
LIN {X -0.5772,Y -135.613,Z 157,A -92.7468,B 24.9683,C -1.3013,E1 25.0013,E2 179.3039} C_DIS
Enddeposition()
LIN {X 0.943,Y -134.6774,Z 157,A -91.845,B 23.1145,C -0.9555,E1 23.1352,E2 179.0183} C_DIS
Startdeposition()
$VEL.CP = VEL_PRINT
LIN {X -2.7538,Y -134.6554,Z 157,A -93.8517,B 23.1153,C -0.9338,E1 23.1294,E2 181.0803} C_DIS
LIN {X -6.3821,Y -134.5317,Z 157,A -95.507,B 23.1156,C -0.9282,E1 23.1248,E2 182.7501} C_DIS
LIN {X -10.4164,Y -134.2805,Z 157,A -97.1975,B 23.1156,C -0.9297,E1 23.1201,E2 184.4377} C_DIS
LIN {X -14.8649,Y -133.8604,Z 157,A -98.9988,B 23.1153,C -0.9347,E1 23.1151,E2 186.2272} C_DIS
LIN {X -17.8969,Y -133.4886,Z 157,A -100.4969,B 23.1157,C -0.9253,E1 23.1109,E2 187.7504} C_DIS
LIN {X -22.089,Y -132.8586,Z 157,A -102.159,B 23.1154,C -0.9327,E1 23.1063,E2 189.3953} C_DIS
LIN {X -25.2875,Y -132.2871,Z 157,A -103.562,B 23.1154,C -0.9322,E1 23.1025,E2 190.8011} C_DIS
LIN {X -28.5909,Y -131.6127,Z 157,A -105.0087,B 23.1154,C -0.9322,E1 23.0985,E2 192.2495} C_DIS
LIN {X -32.7248,Y -130.6467,Z 157,A -106.8536,B 23.1154,C -0.9314,E1 23.0935,E2 194.0995} C_DIS
LIN {X -36.2676,Y -129.7072,Z 157,A -108.3491,B 23.1153,C -0.9355,E1 23.0895,E2 195.587} C_DIS
LIN {X -39.4193,Y -128.7843,Z 157,A -109.7641,B 23.1153,C -0.9356,E1 23.0857,E2 197.0043} C_DIS
LIN {X -43.268,Y -127.545,Z 157,A -111.5193,B 23.1153,C -0.9353,E1 23.081,E2 198.7638} C_DIS
LIN {X -47.5269,Y -126.018,Z 157,A -113.3996,B 23.1151,C -0.9392,E1 23.0761,E2 200.6383} C_DIS
LIN {X -50.562,Y -124.831,Z 157,A -114.7987,B 23.1151,C -0.94,E1 23.0725,E2 202.0387} C_DIS
LIN {X -53.6981,Y -123.5145,Z 157,A -116.2504,B 23.1151,C -0.9413,E1 23.0687,E2 203.4907} C_DIS
LIN {X -57.0622,Y -121.9979,Z 157,A -117.8154,B 23.115,C -0.9434,E1 23.0648,E2 205.0547} C_DIS
LIN {X -59.9128,Y -120.6227,Z 157,A -119.2509,B 23.115,C -0.9408,E1 23.0611,E2 206.5007} C_DIS
LIN {X -64.0143,Y -118.4991,Z 157,A -121.3114,B 23.1151,C -0.9389,E1 23.056,E2 208.5725} C_DIS
LIN {X -67.7551,Y -116.4007,Z 157,A -123.7661,B 23.1162,C -0.9122,E1 23.0499,E2 211.1035} C_DIS
LIN {X -72.7182,Y -113.366,Z 157,A -125.4889,B 23.1147,C -0.951,E1 23.0461,E2 212.733} C_DIS
LIN {X -76.0836,Y -111.1354,Z 157,A -127.287,B 23.1147,C -0.95,E1 23.0419,E2 214.5401} C_DIS
LIN {X -79.7785,Y -108.5134,Z 157,A -129.2174,B 23.1146,C -0.9532,E1 23.0375,E2 216.4697} C_DIS
LIN {X -83.4613,Y -105.7076,Z 157,A -131.2114,B 23.1145,C -0.9557,E1 23.0331,E2 218.4653} C_DIS
LIN {X -86.9324,Y -102.8721,Z 157,A -133.1278,B 23.1144,C -0.9589,E1 23.029,E2 220.3816} C_DIS
LIN {X -90.2177,Y -100.0034,Z 157,A -134.9857,B 23.1142,C -0.9625,E1 23.0251,E2 222.2383} C_DIS
LIN {X -93.4197,Y -97.0189,Z 157,A -136.8868,B 23.1142,C -0.9646,E1 23.0213,E2 224.1426} C_DIS
LIN {X -96.5766,Y -93.8765,Z 157,A -138.78,B 23.114,C -0.9687,E1 23.0175,E2 226.0339} C_DIS
LIN {X -99.7686,Y -90.4764,Z 157,A -140.7366,B 23.1138,C -0.9744,E1 23.0138,E2 227.9853} C_DIS
LIN {X -102.8476,Y -86.9612,Z 157,A -142.7344,B 23.1136,C -0.9786,E1 23.0102,E2 229.9824} C_DIS
LIN {X -105.8679,Y -83.2572,Z 157,A -144.9398,B 23.1137,C -0.9756,E1 23.0063,E2 232.2067} C_DIS
LIN {X -108.7806,Y -79.4147,Z 157,A -146.8761,B 23.1133,C -0.9859,E1 23.0031,E2 234.1268} C_DIS
LIN {X -111.3448,Y -75.7774,Z 157,A -148.7932,B 23.1131,C -0.9897,E1 23.0001,E2 236.0446} C_DIS
LIN {X -113.9099,Y -71.8631,Z 157,A -150.7391,B 23.1128,C -0.997,E1 22.9971,E2 237.9826} C_DIS
LIN {X -116.2553,Y -68.0039,Z 157,A -152.6958,B 23.1128,C -1.0005,E1 22.9943,E2 239.9413} C_DIS
LIN {X -118.4797,Y -64.0505,Z 157,A -154.6225,B 23.1125,C -1.0059,E1 22.9917,E2 241.8651} C_DIS
LIN {X -120.2622,Y -60.6342,Z 157,A -156.1796,B 23.1121,C -1.0143,E1 22.9898,E2 243.41} C_DIS
LIN {X -122.0146,Y -57.0262,Z 157,A -158.2946,B 23.1127,C -1.0006,E1 22.9872,E2 245.5725} C_DIS
LIN {X -123.527,Y -53.6692,Z 157,A -159.2479,B 23.1114,C -1.0329,E1 22.9862,E2 246.4488} C_DIS
LIN {X -124.937,Y -50.299,Z 157,A -161.0581,B 23.1117,C -1.0258,E1 22.9842,E2 248.2881} C_DIS
LIN {X -126.2054,Y -47.0266,Z 157,A -162.5394,B 23.1114,C -1.0308,E1 22.9828,E2 249.7658} C_DIS
LIN {X -127.2823,Y -44.0284,Z 157,A -163.8999,B 23.1113,C -1.0346,E1 22.9815,E2 251.125} C_DIS
LIN {X -128.3299,Y -40.8744,Z 157,A -165.3358,B 23.1111,C -1.0379,E1 22.9803,E2 252.5614} C_DIS
LIN {X -129.4566,Y -37.159,Z 157,A -167.2848,B 23.1115,C -1.0295,E1 22.9787,E2 254.5442} C_DIS
LIN {X -130.9051,Y -31.673,Z 157,A -170.2289,B 23.1122,C -1.0134,E1 22.9767,E2 257.5483} C_DIS
LIN {X -132.175,Y -25.8736,Z 157,A -172.2339,B 23.1109,C -1.0444,E1 22.9756,E2 259.4867} C_DIS
LIN {X -133.1208,Y -20.4504,Z 157,A -174.3576,B 23.1101,C -1.0616,E1 22.9747,E2 261.5802} C_DIS
LIN {X -133.6923,Y -16.305,Z 157,A -176.1583,B 23.1099,C -1.0664,E1 22.974,E2 263.3803} C_DIS
LIN {X -134.0868,Y -12.6546,Z 157,A -177.6945,B 23.1096,C -1.0726,E1 22.9736,E2 264.9108} C_DIS
LIN {X -134.3998,Y -8.733,Z 157,A -179.4462,B 23.1096,C -1.0745,E1 22.9732,E2 266.6692} C_DIS
LIN {X -134.5927,Y -4.9279,Z 157,A 178.8735,B 23.1095,C -1.077,E1 22.973,E2 268.3538} C_DIS
LIN {X -134.6824,Y -0.5735,Z 157,A 177.0715,B 23.1091,C -1.0853,E1 22.973,E2 270.1466} C_DIS
LIN {X -134.6336,Y 3.6329,Z 157,A 175.2839,B 23.1088,C -1.0912,E1 22.973,E2 271.9307} C_DIS
LIN {X -134.4903,Y 7.2065,Z 157,A 173.6515,B 23.1088,C -1.0912,E1 22.9733,E2 273.5739} C_DIS
LIN {X -134.2047,Y 11.3339,Z 157,A 171.9828,B 23.1084,C -1.101,E1 22.9736,E2 275.2285} C_DIS
LIN {X -133.8745,Y 14.7334,Z 157,A 170.4589,B 23.1084,C -1.1026,E1 22.9741,E2 276.7583} C_DIS
LIN {X -133.3467,Y 18.9209,Z 157,A 168.7326,B 23.1079,C -1.1115,E1 22.9747,E2 278.473} C_DIS
LIN {X -132.835,Y 22.2304,Z 157,A 167.2997,B 23.1077,C -1.1157,E1 22.9753,E2 279.9044} C_DIS
LIN {X -132.2437,Y 25.5141,Z 157,A 165.8296,B 23.1077,C -1.118,E1 22.9761,E2 281.3781} C_DIS
LIN {X -130.7411,Y 32.3528,Z 157,A 162.8842,B 23.1071,C -1.129,E1 22.9779,E2 284.3142} C_DIS
LIN {X -129.1352,Y 38.2565,Z 157,A 160.3438,B 23.1066,C -1.1401,E1 22.9798,E2 286.8423} C_DIS
LIN {X -127.4358,Y 43.5855,Z 157,A 157.9578,B 23.1063,C -1.1472,E1 22.9818,E2 289.2249} C_DIS
LIN {X -126.042,Y 47.4629,Z 157,A 156.0747,B 23.1063,C -1.1469,E1 22.9836,E2 291.1206} C_DIS
LIN {X -124.7935,Y 50.655,Z 157,A 154.6099,B 23.1061,C -1.1511,E1 22.9851,E2 292.5836} C_DIS
LIN {X -123.5265,Y 53.6703,Z 157,A 153.2174,B 23.1059,C -1.1553,E1 22.9867,E2 293.9737} C_DIS
LIN {X -122.1289,Y 56.7789,Z 157,A 151.7374,B 23.1057,C -1.1583,E1 22.9884,E2 295.4548} C_DIS
LIN {X -120.6012,Y 59.9563,Z 157,A 150.2222,B 23.1056,C -1.1621,E1 22.9902,E2 296.9692} C_DIS
LIN {X -118.816,Y 63.4244,Z 157,A 148.4433,B 23.1056,C -1.1616,E1 22.9926,E2 298.7596} C_DIS
LIN {X -116.5842,Y 67.438,Z 157,A 146.5149,B 23.1053,C -1.1685,E1 22.9952,E2 300.6815} C_DIS
LIN {X -114.244,Y 71.3311,Z 157,A 144.5878,B 23.105,C -1.1742,E1 22.998,E2 302.6046} C_DIS
LIN {X -111.8772,Y 74.9888,Z 157,A 142.6965,B 23.1048,C -1.1777,E1 23.0009,E2 304.4973} C_DIS
LIN {X -109.3031,Y 78.6941,Z 157,A 140.7419,B 23.1046,C -1.1814,E1 23.0041,E2 306.4529} C_DIS
LIN {X -105.0386,Y 84.3016,Z 157,A 137.9012,B 23.1039,C -1.1965,E1 23.0089,E2 309.2698} C_DIS
LIN {X -102.7916,Y 87.0272,Z 157,A 135.9873,B 23.1046,C -1.1819,E1 23.0124,E2 311.2307} C_DIS
LIN {X -100.4797,Y 89.6863,Z 157,A 134.1258,B 23.1052,C -1.1694,E1 23.0159,E2 313.133} C_DIS
LIN {X -96.822,Y 93.623,Z 157,A 132.4287,B 23.1036,C -1.2016,E1 23.0191,E2 314.756} C_DIS
LIN {X -91.4777,Y 98.8521,Z 157,A 128.5877,B 23.1047,C -1.1793,E1 23.027,E2 318.6711} C_DIS
LIN {X -87.3108,Y 102.5504,Z 157,A 126.8618,B 23.103,C -1.2138,E1 23.0305,E2 320.3163} C_DIS
LIN {X -81.3098,Y 107.371,Z 157,A 123.3155,B 23.1033,C -1.2084,E1 23.0383,E2 323.8905} C_DIS
LIN {X -78.4995,Y 109.4424,Z 157,A 122.0841,B 23.1026,C -1.223,E1 23.041,E2 325.0893} C_DIS
LIN {X -74.9371,Y 111.9117,Z 157,A 120.2084,B 23.1025,C -1.2252,E1 23.0454,E2 326.9662} C_DIS
LIN {X -70.8089,Y 114.5685,Z 157,A 117.9342,B 23.1027,C -1.2207,E1 23.0508,E2 329.26} C_DIS
LIN {X -66.1973,Y 117.2934,Z 157,A 115.8379,B 23.1021,C -1.2331,E1 23.0558,E2 331.3313} C_DIS
LIN {X -62.4965,Y 119.3039,Z 157,A 114.127,B 23.1017,C -1.2399,E1 23.06,E2 333.0301} C_DIS
LIN {X -59.5167,Y 120.8181,Z 157,A 112.6827,B 23.1017,C -1.2411,E1 23.0636,E2 334.4754} C_DIS
LIN {X -56.3746,Y 122.3159,Z 157,A 111.2061,B 23.1015,C -1.2436,E1 23.0673,E2 335.9497} C_DIS
LIN {X -53.3285,Y 123.6743,Z 157,A 109.8013,B 23.1015,C -1.2463,E1 23.0709,E2 337.3512} C_DIS
LIN {X -50.1778,Y 124.9859,Z 157,A 108.3428,B 23.1013,C -1.248,E1 23.0747,E2 338.8089} C_DIS
LIN {X -47.1625,Y 126.1545,Z 157,A 106.9791,B 23.1012,C -1.2504,E1 23.0782,E2 340.1696} C_DIS
LIN {X -43.9821,Y 127.2983,Z 157,A 105.5144,B 23.1012,C -1.251,E1 23.0821,E2 341.6361} C_DIS
LIN {X -40.8135,Y 128.3494,Z 157,A 104.0635,B 23.1012,C -1.2512,E1 23.0859,E2 343.0893} C_DIS
LIN {X -36.7793,Y 129.5641,Z 157,A 102.3985,B 23.1008,C -1.2591,E1 23.0903,E2 344.7372} C_DIS
LIN {X -34.3548,Y 130.2274,Z 157,A 101.2125,B 23.101,C -1.2547,E1 23.0936,E2 345.9363} C_DIS
LIN {X -30.3072,Y 131.2284,Z 157,A 99.4114,B 23.101,C -1.2551,E1 23.0985,E2 347.7391} C_DIS
LIN {X -26.8695,Y 131.9748,Z 157,A 97.9743,B 23.1008,C -1.2591,E1 23.1024,E2 349.1677} C_DIS
LIN {X -23.7324,Y 132.5749,Z 157,A 96.5993,B 23.1008,C -1.2594,E1 23.1062,E2 350.5436} C_DIS
LIN {X -20.4011,Y 133.1284,Z 157,A 95.1119,B 23.1008,C -1.258,E1 23.1103,E2 352.0361} C_DIS
LIN {X -16.145,Y 133.7113,Z 157,A 93.2882,B 23.1008,C -1.2593,E1 23.1153,E2 353.858} C_DIS
LIN {X -12.4913,Y 134.1025,Z 157,A 91.7,B 23.1008,C -1.2588,E1 23.1197,E2 355.4482} C_DIS
LIN {X -8.3369,Y 134.4242,Z 157,A 89.9524,B 23.1007,C -1.2608,E1 23.1246,E2 357.1916} C_DIS
LIN {X -4.1771,Y 134.6185,Z 157,A 88.1383,B 23.1007,C -1.2593,E1 23.1297,E2 359.01} C_DIS
LIN {X -0.5041,Y 134.6819,Z 157,A 86.5466,B 23.1007,C -1.2582,E1 23.1341,E2 360.6044} C_DIS
LIN {X 3.7427,Y 134.6305,Z 157,A 84.8065,B 23.1007,C -1.2616,E1 23.1389,E2 362.3355} C_DIS
LIN {X 7.9593,Y 134.4475,Z 157,A 82.9965,B 23.1007,C -1.2609,E1 23.144,E2 364.1466} C_DIS
LIN {X 11.6346,Y 134.1793,Z 157,A 81.3593,B 23.1008,C -1.2575,E1 23.1486,E2 365.7917} C_DIS
LIN {X 15.8843,Y 133.7424,Z 157,A 79.6439,B 23.1006,C -1.2621,E1 23.1533,E2 367.494} C_DIS
LIN {X 19.4108,Y 133.2767,Z 157,A 78.0126,B 23.1009,C -1.256,E1 23.1579,E2 369.1393} C_DIS
LIN {X 23.6301,Y 132.5932,Z 157,A 76.3254,B 23.1006,C -1.2616,E1 23.1625,E2 370.8102} C_DIS
LIN {X 26.9883,Y 131.9506,Z 157,A 74.8968,B 23.1006,C -1.2622,E1 23.1664,E2 372.2354} C_DIS
LIN {X 30.1763,Y 131.2583,Z 157,A 73.4989,B 23.1006,C -1.261,E1 23.1702,E2 373.6344} C_DIS
LIN {X 33.1176,Y 130.547,Z 157,A 72.1967,B 23.1007,C -1.2595,E1 23.1737,E2 374.9383} C_DIS
LIN {X 36.4134,Y 129.6664,Z 157,A 70.7828,B 23.1007,C -1.2603,E1 23.1775,E2 376.3476} C_DIS
LIN {X 40.2183,Y 128.5395,Z 157,A 68.9661,B 23.1011,C -1.2527,E1 23.1824,E2 378.1802} C_DIS
LIN {X 44.7727,Y 127.0242,Z 157,A 67.0567,B 23.1008,C -1.2574,E1 23.1874,E2 380.0735} C_DIS
LIN {X 47.3351,Y 126.0899,Z 157,A 65.8414,B 23.101,C -1.2536,E1 23.1906,E2 381.2956} C_DIS
LIN {X 51.1315,Y 124.6014,Z 157,A 63.93,B 23.1016,C -1.2431,E1 23.1956,E2 383.2291} C_DIS
LIN {X 55.1765,Y 122.8611,Z 157,A 62.2754,B 23.1011,C -1.2518,E1 23.1998,E2 384.8572} C_DIS
LIN {X 58.2475,Y 121.4352,Z 157,A 60.7973,B 23.1013,C -1.2482,E1 23.2035,E2 386.3403} C_DIS
LIN {X 61.8536,Y 119.6414,Z 157,A 58.9662,B 23.1017,C -1.2401,E1 23.2081,E2 388.1866} C_DIS
LIN {X 66.233,Y 117.2733,Z 157,A 56.5402,B 23.1026,C -1.2219,E1 23.2141,E2 390.651} C_DIS
LIN {X 69.8407,Y 115.1611,Z 157,A 55.2034,B 23.1017,C -1.241,E1 23.2172,E2 391.9346} C_DIS
LIN {X 73.3851,Y 112.9354,Z 157,A 53.3715,B 23.102,C -1.2356,E1 23.2215,E2 393.7738} C_DIS
LIN {X 77.202,Y 110.3618,Z 157,A 51.4266,B 23.102,C -1.233,E1 23.226,E2 395.7181} C_DIS
LIN {X 80.5577,Y 107.9363,Z 157,A 49.6652,B 23.1022,C -1.2299,E1 23.23,E2 397.4807} C_DIS
LIN {X 83.9748,Y 105.2996,Z 157,A 47.5997,B 23.103,C -1.215,E1 23.2346,E2 399.5755} C_DIS
LIN {X 86.6458,Y 103.1129,Z 157,A 46.3933,B 23.1025,C -1.2252,E1 23.2371,E2 400.7508} C_DIS
LIN {X 89.9819,Y 100.215,Z 157,A 44.5209,B 23.1026,C -1.2218,E1 23.241,E2 402.6238} C_DIS
LIN {X 93.2983,Y 97.1355,Z 157,A 42.6002,B 23.1028,C -1.218,E1 23.2449,E2 404.5456} C_DIS
LIN {X 96.458,Y 93.9989,Z 157,A 40.6748,B 23.1031,C -1.2123,E1 23.2487,E2 406.4764} C_DIS
LIN {X 99.5294,Y 90.7401,Z 157,A 38.8123,B 23.1032,C -1.2102,E1 23.2522,E2 408.3355} C_DIS
LIN {X 102.3983,Y 87.4898,Z 157,A 36.9544,B 23.1035,C -1.2052,E1 23.2557,E2 410.1969} C_DIS
LIN {X 105.2203,Y 84.0745,Z 157,A 35.1332,B 23.1035,C -1.2039,E1 23.2589,E2 412.0122} C_DIS
LIN {X 107.7484,Y 80.8096,Z 157,A 33.3237,B 23.1039,C -1.1968,E1 23.2619,E2 413.8301} C_DIS
LIN {X 110.3107,Y 77.2754,Z 157,A 31.1223,B 23.105,C -1.1746,E1 23.2656,E2 416.076} C_DIS
LIN {X 112.6707,Y 73.7914,Z 157,A 30.002,B 23.1035,C -1.2041,E1 23.2672,E2 417.1157} C_DIS
LIN {X 115.4333,Y 69.3905,Z 157,A 27.5086,B 23.1045,C -1.1837,E1 23.2709,E2 419.6469} C_DIS
LIN {X 117.8988,Y 65.1127,Z 157,A 25.3547,B 23.1049,C -1.1752,E1 23.2739,E2 421.8101} C_DIS
LIN {X 122.1649,Y 56.7011,Z 157,A 21.7935,B 23.1044,C -1.1871,E1 23.2783,E2 425.3205} C_DIS
LIN {X 123.7108,Y 53.244,Z 157,A 19.953,B 23.1052,C -1.1706,E1 23.2804,E2 427.1919} C_DIS
LIN {X 125.0192,Y 50.0952,Z 157,A 18.5176,B 23.1053,C -1.1671,E1 23.2819,E2 428.6275} C_DIS
LIN {X 126.2422,Y 46.9284,Z 157,A 17.0059,B 23.1057,C -1.1593,E1 23.2834,E2 430.1497} C_DIS
LIN {X 127.893,Y 42.2228,Z 157,A 15.0138,B 23.1057,C -1.1596,E1 23.2852,E2 432.1289} C_DIS
LIN {X 129.5226,Y 36.9275,Z 157,A 12.6866,B 23.1059,C -1.1539,E1 23.2871,E2 434.456} C_DIS
LIN {X 130.595,Y 32.9286,Z 157,A 10.8982,B 23.1063,C -1.1471,E1 23.2883,E2 436.2505} C_DIS
LIN {X 131.3667,Y 29.7018,Z 157,A 9.4908,B 23.1065,C -1.1429,E1 23.2892,E2 437.6596} C_DIS
LIN {X 132.0584,Y 26.4585,Z 157,A 7.9781,B 23.1069,C -1.1332,E1 23.2901,E2 439.1873} C_DIS
LIN {X 132.8213,Y 22.3125,Z 157,A 6.2618,B 23.1069,C -1.1315,E1 23.2909,E2 440.8969} C_DIS
LIN {X 133.3943,Y 18.588,Z 157,A 4.5933,B 23.1074,C -1.123,E1 23.2916,E2 442.5762} C_DIS
LIN {X 133.8998,Y 14.4983,Z 157,A 2.9265,B 23.1074,C -1.1218,E1 23.2921,E2 444.2352} C_DIS
LIN {X 134.2697,Y 10.5641,Z 157,A 1.1609,B 23.1079,C -1.112,E1 23.2926,E2 446.0142} C_DIS
LIN {X 134.5205,Y 6.605,Z 157,A -0.4102,B 23.1079,C -1.1126,E1 23.2928,E2 447.5736} C_DIS
LIN {X 134.6606,Y 2.4392,Z 157,A -2.1722,B 23.1081,C -1.1074,E1 23.2929,E2 449.3373} C_DIS
LIN {X 134.6746,Y -1.6021,Z 157,A -3.9643,B 23.1085,C -1.098,E1 23.2929,E2 451.1415} C_DIS
LIN {X 134.5707,Y -5.4927,Z 157,A -5.5273,B 23.1085,C -1.0975,E1 23.2928,E2 452.6959} C_DIS
LIN {X 134.3354,Y -9.6641,Z 157,A -7.2981,B 23.1088,C -1.092,E1 23.2925,E2 454.469} C_DIS
LIN {X 134.0185,Y -13.3663,Z 157,A -8.9567,B 23.1092,C -1.0828,E1 23.292,E2 456.1401} C_DIS
LIN {X 133.5476,Y -17.447,Z 157,A -10.5778,B 23.1092,C -1.0837,E1 23.2915,E2 457.7486} C_DIS
LIN {X 133.0065,Y -21.1882,Z 157,A -12.294,B 23.1096,C -1.0728,E1 23.2908,E2 459.4812} C_DIS
LIN {X 132.3047,Y -25.1953,Z 157,A -13.8699,B 23.1096,C -1.0753,E1 23.29,E2 461.0408} C_DIS
LIN {X 131.6484,Y -28.4254,Z 157,A -15.2502,B 23.1096,C -1.0719,E1 23.2892,E2 462.4208} C_DIS
LIN {X 130.9041,Y -31.677,Z 157,A -16.6727,B 23.1099,C -1.0672,E1 23.2883,E2 463.8464} C_DIS
LIN {X 130.0545,Y -35.0031,Z 157,A -18.1446,B 23.1101,C -1.0619,E1 23.2872,E2 465.3224} C_DIS
LIN {X 128.9436,Y -38.8988,Z 157,A -20,B 23.1106,C -1.0496,E1 23.2858,E2 467.1975} C_DIS
LIN {X 127.6762,Y -42.874,Z 157,A -21.5467,B 23.1104,C -1.0558,E1 23.2844,E2 468.7188} C_DIS
LIN {X 126.6178,Y -45.9049,Z 157,A -22.9608,B 23.1107,C -1.049,E1 23.2831,E2 470.1414} C_DIS
LIN {X 125.2368,Y -49.5545,Z 157,A -25.3789,B 23.1125,C -1.0047,E1 23.2805,E2 472.6571} C_DIS
LIN {X 123.0318,Y -54.7949,Z 157,A -26.7723,B 23.1106,C -1.0503,E1 23.2791,E2 473.9268} C_DIS
LIN {X 121.3485,Y -58.4291,Z 157,A -28.6921,B 23.1113,C -1.0339,E1 23.2768,E2 475.8768} C_DIS
LIN {X 119.8727,Y -61.3993,Z 157,A -30.1421,B 23.1116,C -1.0276,E1 23.275,E2 477.3343} C_DIS
LIN {X 117.877,Y -65.152,Z 157,A -32.0034,B 23.1119,C -1.0195,E1 23.2725,E2 479.2056} C_DIS
LIN {X 115.652,Y -69.0246,Z 157,A -33.8722,B 23.1121,C -1.0156,E1 23.2699,E2 481.0737} C_DIS
LIN {X 113.255,Y -72.8915,Z 157,A -35.7964,B 23.1123,C -1.0106,E1 23.267,E2 483} C_DIS
LIN {X 110.8108,Y -76.5566,Z 157,A -37.8154,B 23.1128,C -0.9979,E1 23.2638,E2 485.0403} C_DIS
LIN {X 107.306,Y -81.3959,Z 157,A -40.0165,B 23.1124,C -1.0085,E1 23.2602,E2 487.203} C_DIS
LIN {X 105.1591,Y -84.1513,Z 157,A -41.6903,B 23.1129,C -0.9948,E1 23.2573,E2 488.903} C_DIS
LIN {X 102.3035,Y -87.6008,Z 157,A -43.5932,B 23.1131,C -0.9899,E1 23.2538,E2 490.8087} C_DIS
LIN {X 99.3397,Y -90.9475,Z 157,A -45.4856,B 23.1133,C -0.9855,E1 23.2503,E2 492.703} C_DIS
LIN {X 95.8007,Y -94.6685,Z 157,A -47.4462,B 23.1131,C -0.9916,E1 23.2465,E2 494.639} C_DIS
LIN {X 93.3819,Y -97.0554,Z 157,A -49.1165,B 23.1137,C -0.9765,E1 23.2431,E2 496.3399} C_DIS
LIN {X 90.0608,Y -100.1444,Z 157,A -51.0102,B 23.1137,C -0.9738,E1 23.2392,E2 498.2321} C_DIS
LIN {X 86.1851,Y -103.4989,Z 157,A -52.8804,B 23.1133,C -0.9848,E1 23.2354,E2 500.0666} C_DIS
LIN {X 82.2051,Y -106.6875,Z 157,A -55.3343,B 23.1141,C -0.9655,E1 23.2299,E2 502.5594} C_DIS
LIN {X 78.6453,Y -109.3381,Z 157,A -57.2243,B 23.1143,C -0.9614,E1 23.2256,E2 504.4524} C_DIS
LIN {X 74.9691,Y -111.8904,Z 157,A -59.1082,B 23.1143,C -0.9586,E1 23.2213,E2 506.3364} C_DIS
LIN {X 71.0192,Y -114.4381,Z 157,A -60.9276,B 23.1142,C -0.9639,E1 23.217,E2 508.136} C_DIS
LIN {X 67.8216,Y -116.3622,Z 157,A -62.6672,B 23.1146,C -0.9533,E1 23.2128,E2 509.8968} C_DIS
LIN {X 64.0163,Y -118.498,Z 157,A -64.5271,B 23.1147,C -0.9498,E1 23.2083,E2 511.7595} C_DIS
Enddeposition()
END
